gfCNCPoint1[13267] = {X 367.8420, Y 88.7408, Z -1.3333, A 0.000, B 0.000, C 0.000 }
gfCNCPoint1[13268] = {X 368.7992, Y 88.4188, Z -1.3333, A 0.000, B 0.000, C 0.000 }
gfCNCPoint1[13269] = {X 369.7143, Y 87.9916, Z -1.3333, A 0.000, B 0.000, C 0.000 }
gfCNCPoint1[13270] = {X 370.5758, Y 87.4644, Z -1.3333, A 0.000, B 0.000, C 0.000 }
gfCNCPoint1[13271] = {X 370.7919, Y 87.2394, Z -1.3333, A 0.000, B 0.000, C 0.000 }
gfCNCPoint1[13272] = {X 370.9033, Y 86.9481, Z -1.3333, A 0.000, B 0.000, C 0.000 }
gfCNCPoint1[13273] = {X 371.0969, Y 85.3932, Z -1.3333, A 0.000, B 0.000, C 0.000 }
gfCNCPoint1[13274] = {X 371.1614, Y 83.8276, Z -1.3333, A 0.000, B 0.000, C 0.000 }
gfCNCPoint1[13275] = {X 371.1611, Y 62.9983, Z -1.3333, A 0.000, B 0.000, C 0.000 }
gfCNCPoint1[13276] = {X 371.0248, Y 62.9840, Z -1.3333, A 0.000, B 0.000, C 0.000 }
gfCNCPoint1[13277] = {X 370.8891, Y 62.9651, Z -1.3333, A 0.000, B 0.000, C 0.000 }
gfCNCPoint1[13278] = {X 369.9694, Y 62.7082, Z -1.3333, A 0.000, B 0.000, C 0.000 }
gfCNCPoint1[13279] = {X 369.1346, Y 62.2446, Z -1.3333, A 0.000, B 0.000, C 0.000 }
gfCNCPoint1[13280] = {X 368.4305, Y 61.5997, Z -1.3333, A 0.000, B 0.000, C 0.000 }
gfCNCPoint1[13281] = {X 367.8955, Y 60.8087, Z -1.3333, A 0.000, B 0.000, C 0.000 }
gfCNCPoint1[13282] = {X 367.5590, Y 59.9151, Z -1.3333, A 0.000, B 0.000, C 0.000 }
gfCNCPoint1[13283] = {X 367.4394, Y 58.9678, Z -1.3333, A 0.000, B 0.000, C 0.000 }
gfCNCPoint1[13284] = {X 367.4393, Y 58.0000, Z -1.3333, A 0.000, B 0.000, C 0.000 }
gfCNCPoint1[13285] = {X 367.5416, Y 57.0921, Z -1.3333, A 0.000, B 0.000, C 0.000 }
gfCNCPoint1[13286] = {X 367.8433, Y 56.2298, Z -1.3333, A 0.000, B 0.000, C 0.000 }
gfCNCPoint1[13287] = {X 368.3294, Y 55.4562, Z -1.3333, A 0.000, B 0.000, C 0.000 }
gfCNCPoint1[13288] = {X 368.9754, Y 54.8101, Z -1.3333, A 0.000, B 0.000, C 0.000 }
gfCNCPoint1[13289] = {X 369.7490, Y 54.3240, Z -1.3333, A 0.000, B 0.000, C 0.000 }
gfCNCPoint1[13290] = {X 370.6114, Y 54.0223, Z -1.3333, A 0.000, B 0.000, C 0.000 }
gfCNCPoint1[13291] = {X 371.5193, Y 53.9200, Z -1.3333, A 0.000, B 0.000, C 0.000 }
gfCNCPoint1[13292] = {X 388.0597, Y 53.9200, Z -1.3333, A 0.000, B 0.000, C 0.000 }
gfCNCPoint1[13293] = {X 388.9676, Y 54.0223, Z -1.3333, A 0.000, B 0.000, C 0.000 }
gfCNCPoint1[13294] = {X 389.8299, Y 54.3240, Z -1.3333, A 0.000, B 0.000, C 0.000 }
gfCNCPoint1[13295] = {X 390.6035, Y 54.8101, Z -1.3333, A 0.000, B 0.000, C 0.000 }
gfCNCPoint1[13296] = {X 391.2496, Y 55.4562, Z -1.3333, A 0.000, B 0.000, C 0.000 }
gfCNCPoint1[13297] = {X 391.7356, Y 56.2298, Z -1.3333, A 0.000, B 0.000, C 0.000 }
gfCNCPoint1[13298] = {X 392.0374, Y 57.0921, Z -1.3333, A 0.000, B 0.000, C 0.000 }
gfCNCPoint1[13299] = {X 392.1397, Y 58.0000, Z -1.3333, A 0.000, B 0.000, C 0.000 }
gfCNCPoint1[13300] = {X 392.1397, Y 58.9342, Z -1.3333, A 0.000, B 0.000, C 0.000 }
gfCNCPoint1[13301] = {X 392.0298, Y 59.8744, Z -1.3333, A 0.000, B 0.000, C 0.000 }
gfCNCPoint1[13302] = {X 391.7063, Y 60.7639, Z -1.3333, A 0.000, B 0.000, C 0.000 }
gfCNCPoint1[13303] = {X 391.1724, Y 61.5726, Z -1.3333, A 0.000, B 0.000, C 0.000 }
gfCNCPoint1[13304] = {X 390.4636, Y 62.2335, Z -1.3333, A 0.000, B 0.000, C 0.000 }
gfCNCPoint1[13305] = {X 389.6195, Y 62.7095, Z -1.3333, A 0.000, B 0.000, C 0.000 }
gfCNCPoint1[13306] = {X 388.6872, Y 62.9742, Z -1.3333, A 0.000, B 0.000, C 0.000 }
gfCNCPoint1[13307] = {X 388.5540, Y 62.9932, Z -1.3333, A 0.000, B 0.000, C 0.000 }
gfCNCPoint1[13308] = {X 388.4202, Y 63.0078, Z -1.3333, A 0.000, B 0.000, C 0.000 }
gfCNCPoint1[13309] = {X 388.4176, Y 63.1548, Z -1.3333, A 0.000, B 0.000, C 0.000 }
gfCNCPoint1[13310] = {X 388.4156, Y 84.6157, Z -1.3333, A 0.000, B 0.000, C 0.000 }
gfCNCPoint1[13311] = {X 388.3564, Y 86.2534, Z -1.3333, A 0.000, B 0.000, C 0.000 }
gfCNCPoint1[13312] = {X 388.1546, Y 87.8797, Z -1.3333, A 0.000, B 0.000, C 0.000 }
gfCNCPoint1[13313] = {X 387.8118, Y 89.4822, Z -1.3333, A 0.000, B 0.000, C 0.000 }
gfCNCPoint1[13314] = {X 387.2905, Y 91.0377, Z -1.3333, A 0.000, B 0.000, C 0.000 }
gfCNCPoint1[13315] = {X 386.5561, Y 92.5046, Z -1.3333, A 0.000, B 0.000, C 0.000 }
gfCNCPoint1[13316] = {X 385.6232, Y 93.8539, Z -1.3333, A 0.000, B 0.000, C 0.000 }
gfCNCPoint1[13317] = {X 384.5101, Y 95.0589, Z -1.3333, A 0.000, B 0.000, C 0.000 }
gfCNCPoint1[13318] = {X 383.0155, Y 96.3179, Z -1.3333, A 0.000, B 0.000, C 0.000 }
gfCNCPoint1[13319] = {X 381.3959, Y 97.4112, Z -1.3333, A 0.000, B 0.000, C 0.000 }
gfCNCPoint1[13320] = {X 379.6694, Y 98.3265, Z -1.3333, A 0.000, B 0.000, C 0.000 }
gfCNCPoint1[13321] = {X 377.4145, Y 99.2771, Z -1.3333, A 0.000, B 0.000, C 0.000 }
gfCNCPoint1[13322] = {X 375.0967, Y 100.0618, Z -1.3333, A 0.000, B 0.000, C 0.000 }
gfCNCPoint1[13323] = {X 372.7281, Y 100.6767, Z -1.3333, A 0.000, B 0.000, C 0.000 }
gfCNCPoint1[13324] = {X 368.9280, Y 101.4118, Z -1.3333, A 0.000, B 0.000, C 0.000 }
gfCNCPoint1[13325] = {X 365.0969, Y 101.9635, Z -1.3333, A 0.000, B 0.000, C 0.000 }
gfCNCPoint1[13326] = {X 361.2438, Y 102.3303, Z -1.3333, A 0.000, B 0.000, C 0.000 }
gfCNCPoint1[13327] = {X 357.2421, Y 102.5707, Z -1.3333, A 0.000, B 0.000, C 0.000 }
gfCNCPoint1[13328] = {X 353.2361, Y 102.7240, Z -1.3333, A 0.000, B 0.000, C 0.000 }
gfCNCPoint1[13329] = {X 353.3455, Y 106.7225, Z -1.3333, A 0.000, B 0.000, C 0.000 }
gfCNCPoint1[13330] = {X 353.2339, Y 102.6440, Z -1.3333, A 0.000, B 0.000, C 0.000 }
gfCNCPoint1[13331] = {X 347.7211, Y 102.7124, Z -1.3333, A 0.000, B 0.000, C 0.000 }
gfCNCPoint1[13332] = {X 342.2087, Y 102.6158, Z -1.3333, A 0.000, B 0.000, C 0.000 }
gfCNCPoint1[13333] = {X 336.7017, Y 102.3544, Z -1.3333, A 0.000, B 0.000, C 0.000 }
gfCNCPoint1[13334] = {X 333.2238, Y 102.0803, Z -1.3333, A 0.000, B 0.000, C 0.000 }
gfCNCPoint1[13335] = {X 329.7596, Y 101.6688, Z -1.3333, A 0.000, B 0.000, C 0.000 }
gfCNCPoint1[13336] = {X 326.3144, Y 101.1205, Z -1.3333, A 0.000, B 0.000, C 0.000 }
gfCNCPoint1[13337] = {X 323.4875, Y 100.5209, Z -1.3333, A 0.000, B 0.000, C 0.000 }
gfCNCPoint1[13338] = {X 320.7125, Y 99.7145, Z -1.3333, A 0.000, B 0.000, C 0.000 }
gfCNCPoint1[13339] = {X 318.0046, Y 98.7056, Z -1.3333, A 0.000, B 0.000, C 0.000 }
gfCNCPoint1[13340] = {X 316.5155, Y 98.0196, Z -1.3333, A 0.000, B 0.000, C 0.000 }
gfCNCPoint1[13341] = {X 315.0892, Y 97.2110, Z -1.3333, A 0.000, B 0.000, C 0.000 }
gfCNCPoint1[13342] = {X 313.7357, Y 96.2857, Z -1.3333, A 0.000, B 0.000, C 0.000 }
gfCNCPoint1[13343] = {X 312.4647, Y 95.2501, Z -1.3333, A 0.000, B 0.000, C 0.000 }
gfCNCPoint1[13344] = {X 311.4884, Y 94.2784, Z -1.3333, A 0.000, B 0.000, C 0.000 }
gfCNCPoint1[13345] = {X 310.6340, Y 93.1980, Z -1.3333, A 0.000, B 0.000, C 0.000 }
gfCNCPoint1[13346] = {X 309.9137, Y 92.0239, Z -1.3333, A 0.000, B 0.000, C 0.000 }
gfCNCPoint1[13347] = {X 309.3376, Y 90.7727, Z -1.3333, A 0.000, B 0.000, C 0.000 }
gfCNCPoint1[13348] = {X 308.9138, Y 89.4621, Z -1.3333, A 0.000, B 0.000, C 0.000 }
gfCNCPoint1[13349] = {X 308.5760, Y 87.8658, Z -1.3333, A 0.000, B 0.000, C 0.000 }
gfCNCPoint1[13350] = {X 308.3765, Y 86.2464, Z -1.3333, A 0.000, B 0.000, C 0.000 }
gfCNCPoint1[13351] = {X 308.3167, Y 84.6159, Z -1.3333, A 0.000, B 0.000, C 0.000 }
gfCNCPoint1[13352] = {X 308.3180, Y 83.2313, Z -1.3333, A 0.000, B 0.000, C 0.000 }
gfCNCPoint1[13353] = {X 308.3180, Y 62.9244, Z -1.3333, A 0.000, B 0.000, C 0.000 }
gfCNCPoint1[13354] = {X 307.4752, Y 62.7738, Z -1.3333, A 0.000, B 0.000, C 0.000 }
gfCNCPoint1[13355] = {X 306.6837, Y 62.4472, Z -1.3333, A 0.000, B 0.000, C 0.000 }
gfCNCPoint1[13356] = {X 305.9799, Y 61.9597, Z -1.3333, A 0.000, B 0.000, C 0.000 }
gfCNCPoint1[13357] = {X 305.3959, Y 61.3336, Z -1.3333, A 0.000, B 0.000, C 0.000 }
gfCNCPoint1[13358] = {X 304.9585, Y 60.5976, Z -1.3333, A 0.000, B 0.000, C 0.000 }
gfCNCPoint1[13359] = {X 304.6878, Y 59.7853, Z -1.3333, A 0.000, B 0.000, C 0.000 }
gfCNCPoint1[13360] = {X 304.5962, Y 58.9340, Z -1.3333, A 0.000, B 0.000, C 0.000 }
gfCNCPoint1[13361] = {X 304.5962, Y 58.0000, Z -1.3333, A 0.000, B 0.000, C 0.000 }
gfCNCPoint1[13362] = {X 304.6965, Y 57.1099, Z -1.3333, A 0.000, B 0.000, C 0.000 }
gfCNCPoint1[13363] = {X 304.9923, Y 56.2645, Z -1.3333, A 0.000, B 0.000, C 0.000 }
gfCNCPoint1[13364] = {X 305.4689, Y 55.5060, Z -1.3333, A 0.000, B 0.000, C 0.000 }
gfCNCPoint1[13365] = {X 306.1023, Y 54.8727, Z -1.3333, A 0.000, B 0.000, C 0.000 }
gfCNCPoint1[13366] = {X 306.8607, Y 54.3961, Z -1.3333, A 0.000, B 0.000, C 0.000 }
gfCNCPoint1[13367] = {X 307.7061, Y 54.1003, Z -1.3333, A 0.000, B 0.000, C 0.000 }
gfCNCPoint1[13368] = {X 308.5962, Y 54.0000, Z -1.3333, A 0.000, B 0.000, C 0.000 }
gfCNCPoint1[13369] = {X 324.3107, Y 54.0000, Z -1.3333, A 0.000, B 0.000, C 0.000 }
gfCNCPoint1[13370] = {X 325.2008, Y 54.1003, Z -1.3333, A 0.000, B 0.000, C 0.000 }
gfCNCPoint1[13371] = {X 326.0462, Y 54.3961, Z -1.3333, A 0.000, B 0.000, C 0.000 }
gfCNCPoint1[13372] = {X 326.8046, Y 54.8727, Z -1.3333, A 0.000, B 0.000, C 0.000 }
gfCNCPoint1[13373] = {X 327.4380, Y 55.5060, Z -1.3333, A 0.000, B 0.000, C 0.000 }
gfCNCPoint1[13374] = {X 327.9146, Y 56.2645, Z -1.3333, A 0.000, B 0.000, C 0.000 }
gfCNCPoint1[13375] = {X 328.2104, Y 57.1099, Z -1.3333, A 0.000, B 0.000, C 0.000 }
gfCNCPoint1[13376] = {X 328.3107, Y 58.0000, Z -1.3333, A 0.000, B 0.000, C 0.000 }
gfCNCPoint1[13377] = {X 328.3107, Y 58.9341, Z -1.3333, A 0.000, B 0.000, C 0.000 }
gfCNCPoint1[13378] = {X 328.2147, Y 59.7843, Z -1.3333, A 0.000, B 0.000, C 0.000 }
gfCNCPoint1[13379] = {X 327.9419, Y 60.5952, Z -1.3333, A 0.000, B 0.000, C 0.000 }
gfCNCPoint1[13380] = {X 327.5044, Y 61.3305, Z -1.3333, A 0.000, B 0.000, C 0.000 }
gfCNCPoint1[13381] = {X 326.9218, Y 61.9572, Z -1.3333, A 0.000, B 0.000, C 0.000 }
gfCNCPoint1[13382] = {X 326.2204, Y 62.4471, Z -1.3333, A 0.000, B 0.000, C 0.000 }
gfCNCPoint1[13383] = {X 325.4315, Y 62.7783, Z -1.3333, A 0.000, B 0.000, C 0.000 }
gfCNCPoint1[13384] = {X 324.5905, Y 62.9360, Z -1.3333, A 0.000, B 0.000, C 0.000 }
gfCNCPoint1[13385] = {X 324.5919, Y 83.2313, Z -1.3333, A 0.000, B 0.000, C 0.000 }
gfCNCPoint1[13386] = {X 324.6054, Y 84.6159, Z -1.3333, A 0.000, B 0.000, C 0.000 }
gfCNCPoint1[13387] = {X 324.6887, Y 85.9184, Z -1.3333, A 0.000, B 0.000, C 0.000 }
gfCNCPoint1[13388] = {X 324.9294, Y 87.2011, Z -1.3333, A 0.000, B 0.000, C 0.000 }
gfCNCPoint1[13389] = {X 325.2359, Y 87.5559, Z -1.3333, A 0.000, B 0.000, C 0.000 }
gfCNCPoint1[13390] = {X 325.6219, Y 87.8220, Z -1.3333, A 0.000, B 0.000, C 0.000 }
gfCNCPoint1[13391] = {X 326.0749, Y 88.0775, Z -1.3333, A 0.000, B 0.000, C 0.000 }
gfCNCPoint1[13392] = {X 327.5502, Y 88.6916, Z -1.3333, A 0.000, B 0.000, C 0.000 }
gfCNCPoint1[13393] = {X 329.0843, Y 89.1390, Z -1.3333, A 0.000, B 0.000, C 0.000 }
gfCNCPoint1[13394] = {X 332.1822, Y 89.7592, Z -1.3333, A 0.000, B 0.000, C 0.000 }
gfCNCPoint1[13395] = {X 335.3167, Y 90.1542, Z -1.3333, A 0.000, B 0.000, C 0.000 }
gfCNCPoint1[13396] = {X 340.5042, Y 90.5381, Z -1.3333, A 0.000, B 0.000, C 0.000 }
gfCNCPoint1[13397] = {X 345.7039, Y 90.6832, Z -1.3333, A 0.000, B 0.000, C 0.000 }
gfCNCPoint1[13398] = {X 350.5564, Y 90.6891, Z -1.3333, A 0.000, B 0.000, C 0.000 }
gfCNCPoint1[13399] = {X 355.4059, Y 90.5203, Z -1.3333, A 0.000, B 0.000, C 0.000 }
gfCNCPoint1[13400] = {X 360.2461, Y 90.1768, Z -1.3333, A 0.000, B 0.000, C 0.000 }
gfCNCPoint1[13401] = {X 362.8123, Y 89.8853, Z -1.3333, A 0.000, B 0.000, C 0.000 }
gfCNCPoint1[13402] = {X 365.3548, Y 89.4317, Z -1.3333, A 0.000, B 0.000, C 0.000 }
gfCNCPoint1[13403] = {X 367.8634, Y 88.8179, Z -1.3333, A 0.000, B 0.000, C 0.000 }
gfCNCPoint1[13404] = {X 368.8291, Y 88.4930, Z -1.3333, A 0.000, B 0.000, C 0.000 }
gfCNCPoint1[13405] = {X 369.7523, Y 88.0620, Z -1.3333, A 0.000, B 0.000, C 0.000 }
gfCNCPoint1[13406] = {X 370.6213, Y 87.5302, Z -1.3333, A 0.000, B 0.000, C 0.000 }
gfCNCPoint1[13407] = {X 370.8594, Y 87.2823, Z -1.3333, A 0.000, B 0.000, C 0.000 }
gfCNCPoint1[13408] = {X 370.9822, Y 86.9612, Z -1.3333, A 0.000, B 0.000, C 0.000 }
gfCNCPoint1[13409] = {X 371.1766, Y 85.3997, Z -1.3333, A 0.000, B 0.000, C 0.000 }
gfCNCPoint1[13410] = {X 371.2414, Y 83.8276, Z -1.3333, A 0.000, B 0.000, C 0.000 }
gfCNCPoint1[13411] = {X 371.2396, Y 63.0383, Z -1.3333, A 0.000, B 0.000, C 0.000 }
gfCNCPoint1[13412] = {X 371.2440, Y 62.9246, Z -1.3333, A 0.000, B 0.000, C 0.000 }
gfCNCPoint1[13413] = {X 371.0723, Y 62.9090, Z -1.3333, A 0.000, B 0.000, C 0.000 }
gfCNCPoint1[13414] = {X 370.9014, Y 62.8861, Z -1.3333, A 0.000, B 0.000, C 0.000 }
gfCNCPoint1[13415] = {X 369.9947, Y 62.6321, Z -1.3333, A 0.000, B 0.000, C 0.000 }
gfCNCPoint1[13416] = {X 369.1724, Y 62.1733, Z -1.3333, A 0.000, B 0.000, C 0.000 }
gfCNCPoint1[13417] = {X 368.4802, Y 61.5349, Z -1.3333, A 0.000, B 0.000, C 0.000 }
gfCNCPoint1[13418] = {X 367.9565, Y 60.7524, Z -1.3333, A 0.000, B 0.000, C 0.000 }
gfCNCPoint1[13419] = {X 367.6301, Y 59.8691, Z -1.3333, A 0.000, B 0.000, C 0.000 }
gfCNCPoint1[13420] = {X 367.5193, Y 58.9340, Z -1.3333, A 0.000, B 0.000, C 0.000 }
gfCNCPoint1[13421] = {X 367.5193, Y 58.0000, Z -1.3333, A 0.000, B 0.000, C 0.000 }
gfCNCPoint1[13422] = {X 367.6196, Y 57.1099, Z -1.3333, A 0.000, B 0.000, C 0.000 }
gfCNCPoint1[13423] = {X 367.9154, Y 56.2645, Z -1.3333, A 0.000, B 0.000, C 0.000 }
gfCNCPoint1[13424] = {X 368.3920, Y 55.5060, Z -1.3333, A 0.000, B 0.000, C 0.000 }
gfCNCPoint1[13425] = {X 369.0253, Y 54.8727, Z -1.3333, A 0.000, B 0.000, C 0.000 }
gfCNCPoint1[13426] = {X 369.7837, Y 54.3961, Z -1.3333, A 0.000, B 0.000, C 0.000 }
gfCNCPoint1[13427] = {X 370.6292, Y 54.1003, Z -1.3333, A 0.000, B 0.000, C 0.000 }
gfCNCPoint1[13428] = {X 371.5193, Y 54.0000, Z -1.3333, A 0.000, B 0.000, C 0.000 }
gfCNCPoint1[13429] = {X 388.0597, Y 54.0000, Z -1.3333, A 0.000, B 0.000, C 0.000 }
gfCNCPoint1[13430] = {X 388.9498, Y 54.1003, Z -1.3333, A 0.000, B 0.000, C 0.000 }
gfCNCPoint1[13431] = {X 389.7952, Y 54.3961, Z -1.3333, A 0.000, B 0.000, C 0.000 }
gfCNCPoint1[13432] = {X 390.5536, Y 54.8727, Z -1.3333, A 0.000, B 0.000, C 0.000 }
gfCNCPoint1[13433] = {X 391.1870, Y 55.5060, Z -1.3333, A 0.000, B 0.000, C 0.000 }
gfCNCPoint1[13434] = {X 391.6636, Y 56.2645, Z -1.3333, A 0.000, B 0.000, C 0.000 }
gfCNCPoint1[13435] = {X 391.9594, Y 57.1099, Z -1.3333, A 0.000, B 0.000, C 0.000 }
gfCNCPoint1[13436] = {X 392.0597, Y 58.0000, Z -1.3333, A 0.000, B 0.000, C 0.000 }
gfCNCPoint1[13437] = {X 392.0595, Y 58.9671, Z -1.3333, A 0.000, B 0.000, C 0.000 }
gfCNCPoint1[13438] = {X 391.9482, Y 59.8719, Z -1.3333, A 0.000, B 0.000, C 0.000 }
gfCNCPoint1[13439] = {X 391.6348, Y 60.7280, Z -1.3333, A 0.000, B 0.000, C 0.000 }
gfCNCPoint1[13440] = {X 391.1113, Y 61.5210, Z -1.3333, A 0.000, B 0.000, C 0.000 }
gfCNCPoint1[13441] = {X 390.4163, Y 62.1689, Z -1.3333, A 0.000, B 0.000, C 0.000 }
gfCNCPoint1[13442] = {X 389.5887, Y 62.6357, Z -1.3333, A 0.000, B 0.000, C 0.000 }
gfCNCPoint1[13443] = {X 388.6746, Y 62.8952, Z -1.3333, A 0.000, B 0.000, C 0.000 }
gfCNCPoint1[13444] = {X 388.5085, Y 62.9182, Z -1.3333, A 0.000, B 0.000, C 0.000 }
gfCNCPoint1[13445] = {X 388.3415, Y 62.9342, Z -1.3333, A 0.000, B 0.000, C 0.000 }
gfCNCPoint1[13446] = {X 388.3376, Y 63.1540, Z -1.3333, A 0.000, B 0.000, C 0.000 }
gfCNCPoint1[13447] = {X 388.3376, Y 83.9236, Z -1.3333, A 0.000, B 0.000, C 0.000 }
gfCNCPoint1[13448] = {X 388.3356, Y 84.6159, Z -1.3333, A 0.000, B 0.000, C 0.000 }
gfCNCPoint1[13449] = {X 388.2766, Y 86.2468, Z -1.3333, A 0.000, B 0.000, C 0.000 }
gfCNCPoint1[13450] = {X 388.0757, Y 87.8663, Z -1.3333, A 0.000, B 0.000, C 0.000 }
gfCNCPoint1[13451] = {X 387.7344, Y 89.4621, Z -1.3333, A 0.000, B 0.000, C 0.000 }
gfCNCPoint1[13452] = {X 387.2167, Y 91.0069, Z -1.3333, A 0.000, B 0.000, C 0.000 }
gfCNCPoint1[13453] = {X 386.4873, Y 92.4638, Z -1.3333, A 0.000, B 0.000, C 0.000 }
gfCNCPoint1[13454] = {X 385.5607, Y 93.8039, Z -1.3333, A 0.000, B 0.000, C 0.000 }
gfCNCPoint1[13455] = {X 384.4553, Y 95.0007, Z -1.3333, A 0.000, B 0.000, C 0.000 }
gfCNCPoint1[13456] = {X 382.9672, Y 96.2541, Z -1.3333, A 0.000, B 0.000, C 0.000 }
gfCNCPoint1[13457] = {X 381.3546, Y 97.3426, Z -1.3333, A 0.000, B 0.000, C 0.000 }
gfCNCPoint1[13458] = {X 379.6357, Y 98.2540, Z -1.3333, A 0.000, B 0.000, C 0.000 }
gfCNCPoint1[13459] = {X 377.3861, Y 99.2023, Z -1.3333, A 0.000, B 0.000, C 0.000 }
gfCNCPoint1[13460] = {X 375.0738, Y 99.9852, Z -1.3333, A 0.000, B 0.000, C 0.000 }
gfCNCPoint1[13461] = {X 372.7108, Y 100.5986, Z -1.3333, A 0.000, B 0.000, C 0.000 }
gfCNCPoint1[13462] = {X 368.9146, Y 101.3330, Z -1.3333, A 0.000, B 0.000, C 0.000 }
gfCNCPoint1[13463] = {X 365.0874, Y 101.8841, Z -1.3333, A 0.000, B 0.000, C 0.000 }
gfCNCPoint1[13464] = {X 361.2381, Y 102.2505, Z -1.3333, A 0.000, B 0.000, C 0.000 }
gfCNCPoint1[13465] = {X 357.2381, Y 102.4908, Z -1.3333, A 0.000, B 0.000, C 0.000 }
gfCNCPoint1[13466] = {X 353.2339, Y 102.6440, Z -1.3333, A 0.000, B 0.000, C 0.000 }
gfCNCPoint1[13467] = {X 353.3455, Y 106.7225, Z -1.3333, A 0.000, B 0.000, C 0.000 }
gfCNCPoint1[13468] = {X 353.3455, Y 106.7225, Z 1.6667, A 0.000, B 0.000, C 0.000 }
gfCNCPoint1[13469] = {X 353.3455, Y 106.7225, Z 11.0000, A 0.000, B 0.000, C 0.000 }
gfCNCPoint1[13470] = {X 411.5994, Y 79.5934, Z 11.0000, A 0.000, B 0.000, C 0.000 }
gfCNCPoint1[13471] = {X 411.5994, Y 79.5934, Z 1.6667, A 0.000, B 0.000, C 0.000 }
gfCNCPoint1[13472] = {X 411.5994, Y 79.5934, Z -1.3333, A 0.000, B 0.000, C 0.000 }
gfCNCPoint1[13473] = {X 413.7997, Y 83.0292, Z -1.3333, A 0.000, B 0.000, C 0.000 }
gfCNCPoint1[13474] = {X 428.0558, Y 73.8994, Z -1.3333, A 0.000, B 0.000, C 0.000 }
gfCNCPoint1[13475] = {X 403.7554, Y 64.3645, Z -1.3333, A 0.000, B 0.000, C 0.000 }
gfCNCPoint1[13476] = {X 402.0597, Y 63.8030, Z -1.3333, A 0.000, B 0.000, C 0.000 }
gfCNCPoint1[13477] = {X 400.3124, Y 63.4313, Z -1.3333, A 0.000, B 0.000, C 0.000 }
gfCNCPoint1[13478] = {X 398.5349, Y 63.2540, Z -1.3333, A 0.000, B 0.000, C 0.000 }
gfCNCPoint1[13479] = {X 397.5823, Y 63.1425, Z -1.3333, A 0.000, B 0.000, C 0.000 }
gfCNCPoint1[13480] = {X 396.6778, Y 62.8236, Z -1.3333, A 0.000, B 0.000, C 0.000 }
gfCNCPoint1[13481] = {X 395.8660, Y 62.3130, Z -1.3333, A 0.000, B 0.000, C 0.000 }
gfCNCPoint1[13482] = {X 395.1868, Y 61.6358, Z -1.3333, A 0.000, B 0.000, C 0.000 }
gfCNCPoint1[13483] = {X 394.6738, Y 60.8255, Z -1.3333, A 0.000, B 0.000, C 0.000 }
gfCNCPoint1[13484] = {X 394.3522, Y 59.9220, Z -1.3333, A 0.000, B 0.000, C 0.000 }
gfCNCPoint1[13485] = {X 394.2379, Y 58.9697, Z -1.3333, A 0.000, B 0.000, C 0.000 }
gfCNCPoint1[13486] = {X 394.2377, Y 58.0000, Z -1.3333, A 0.000, B 0.000, C 0.000 }
gfCNCPoint1[13487] = {X 394.3460, Y 57.0387, Z -1.3333, A 0.000, B 0.000, C 0.000 }
gfCNCPoint1[13488] = {X 394.6655, Y 56.1256, Z -1.3333, A 0.000, B 0.000, C 0.000 }
gfCNCPoint1[13489] = {X 395.1802, Y 55.3065, Z -1.3333, A 0.000, B 0.000, C 0.000 }
gfCNCPoint1[13490] = {X 395.8642, Y 54.6225, Z -1.3333, A 0.000, B 0.000, C 0.000 }
gfCNCPoint1[13491] = {X 396.6833, Y 54.1078, Z -1.3333, A 0.000, B 0.000, C 0.000 }
gfCNCPoint1[13492] = {X 397.5964, Y 53.7883, Z -1.3333, A 0.000, B 0.000, C 0.000 }
gfCNCPoint1[13493] = {X 398.5577, Y 53.6800, Z -1.3333, A 0.000, B 0.000, C 0.000 }
gfCNCPoint1[13494] = {X 419.4886, Y 53.6800, Z -1.3333, A 0.000, B 0.000, C 0.000 }
gfCNCPoint1[13495] = {X 420.4499, Y 53.7883, Z -1.3333, A 0.000, B 0.000, C 0.000 }
gfCNCPoint1[13496] = {X 421.3630, Y 54.1078, Z -1.3333, A 0.000, B 0.000, C 0.000 }
gfCNCPoint1[13497] = {X 422.1821, Y 54.6225, Z -1.3333, A 0.000, B 0.000, C 0.000 }
gfCNCPoint1[13498] = {X 422.8661, Y 55.3065, Z -1.3333, A 0.000, B 0.000, C 0.000 }
gfCNCPoint1[13499] = {X 423.3808, Y 56.1256, Z -1.3333, A 0.000, B 0.000, C 0.000 }
gfCNCPoint1[13500] = {X 423.7003, Y 57.0387, Z -1.3333, A 0.000, B 0.000, C 0.000 }
gfCNCPoint1[13501] = {X 423.8086, Y 58.0000, Z -1.3333, A 0.000, B 0.000, C 0.000 }
gfCNCPoint1[13502] = {X 423.8086, Y 58.2329, Z -1.3333, A 0.000, B 0.000, C 0.000 }
gfCNCPoint1[13503] = {X 429.6116, Y 60.4947, Z -1.3333, A 0.000, B 0.000, C 0.000 }
gfCNCPoint1[13504] = {X 457.8614, Y 71.7026, Z -1.3333, A 0.000, B 0.000, C 0.000 }
gfCNCPoint1[13505] = {X 457.8614, Y 63.2124, Z -1.3333, A 0.000, B 0.000, C 0.000 }
gfCNCPoint1[13506] = {X 457.0096, Y 63.0035, Z -1.3333, A 0.000, B 0.000, C 0.000 }
gfCNCPoint1[13507] = {X 456.2176, Y 62.6267, Z -1.3333, A 0.000, B 0.000, C 0.000 }
gfCNCPoint1[13508] = {X 455.5180, Y 62.0978, Z -1.3333, A 0.000, B 0.000, C 0.000 }
gfCNCPoint1[13509] = {X 454.9396, Y 61.4384, Z -1.3333, A 0.000, B 0.000, C 0.000 }
gfCNCPoint1[13510] = {X 454.5063, Y 60.6759, Z -1.3333, A 0.000, B 0.000, C 0.000 }
gfCNCPoint1[13511] = {X 454.2360, Y 59.8415, Z -1.3333, A 0.000, B 0.000, C 0.000 }
gfCNCPoint1[13512] = {X 454.1398, Y 58.9697, Z -1.3333, A 0.000, B 0.000, C 0.000 }
gfCNCPoint1[13513] = {X 454.1396, Y 58.0000, Z -1.3333, A 0.000, B 0.000, C 0.000 }
gfCNCPoint1[13514] = {X 454.2479, Y 57.0387, Z -1.3333, A 0.000, B 0.000, C 0.000 }
gfCNCPoint1[13515] = {X 454.5674, Y 56.1256, Z -1.3333, A 0.000, B 0.000, C 0.000 }
gfCNCPoint1[13516] = {X 455.0821, Y 55.3065, Z -1.3333, A 0.000, B 0.000, C 0.000 }
gfCNCPoint1[13517] = {X 455.7661, Y 54.6225, Z -1.3333, A 0.000, B 0.000, C 0.000 }
gfCNCPoint1[13518] = {X 456.5852, Y 54.1078, Z -1.3333, A 0.000, B 0.000, C 0.000 }
gfCNCPoint1[13519] = {X 457.4983, Y 53.7883, Z -1.3333, A 0.000, B 0.000, C 0.000 }
gfCNCPoint1[13520] = {X 458.4596, Y 53.6800, Z -1.3333, A 0.000, B 0.000, C 0.000 }
gfCNCPoint1[13521] = {X 475.0000, Y 53.6800, Z -1.3333, A 0.000, B 0.000, C 0.000 }
gfCNCPoint1[13522] = {X 475.9613, Y 53.7883, Z -1.3333, A 0.000, B 0.000, C 0.000 }
gfCNCPoint1[13523] = {X 476.8744, Y 54.1078, Z -1.3333, A 0.000, B 0.000, C 0.000 }
gfCNCPoint1[13524] = {X 477.6935, Y 54.6225, Z -1.3333, A 0.000, B 0.000, C 0.000 }
gfCNCPoint1[13525] = {X 478.3775, Y 55.3065, Z -1.3333, A 0.000, B 0.000, C 0.000 }
gfCNCPoint1[13526] = {X 478.8922, Y 56.1256, Z -1.3333, A 0.000, B 0.000, C 0.000 }
gfCNCPoint1[13527] = {X 479.2117, Y 57.0387, Z -1.3333, A 0.000, B 0.000, C 0.000 }
gfCNCPoint1[13528] = {X 479.3200, Y 58.0000, Z -1.3333, A 0.000, B 0.000, C 0.000 }
gfCNCPoint1[13529] = {X 479.3200, Y 58.9342, Z -1.3333, A 0.000, B 0.000, C 0.000 }
gfCNCPoint1[13530] = {X 479.2299, Y 59.8116, Z -1.3333, A 0.000, B 0.000, C 0.000 }
gfCNCPoint1[13531] = {X 478.9636, Y 60.6524, Z -1.3333, A 0.000, B 0.000, C 0.000 }
gfCNCPoint1[13532] = {X 478.5320, Y 61.4215, Z -1.3333, A 0.000, B 0.000, C 0.000 }
gfCNCPoint1[13533] = {X 477.9532, Y 62.0870, Z -1.3333, A 0.000, B 0.000, C 0.000 }
gfCNCPoint1[13534] = {X 477.2513, Y 62.6211, Z -1.3333, A 0.000, B 0.000, C 0.000 }
gfCNCPoint1[13535] = {X 476.4556, Y 63.0014, Z -1.3333, A 0.000, B 0.000, C 0.000 }
gfCNCPoint1[13536] = {X 475.5992, Y 63.2123, Z -1.3333, A 0.000, B 0.000, C 0.000 }
gfCNCPoint1[13537] = {X 475.5996, Y 92.7691, Z -1.3333, A 0.000, B 0.000, C 0.000 }
gfCNCPoint1[13538] = {X 475.9955, Y 92.8681, Z -1.3333, A 0.000, B 0.000, C 0.000 }
gfCNCPoint1[13539] = {X 476.3859, Y 92.9874, Z -1.3333, A 0.000, B 0.000, C 0.000 }
gfCNCPoint1[13540] = {X 477.1980, Y 93.3562, Z -1.3333, A 0.000, B 0.000, C 0.000 }
gfCNCPoint1[13541] = {X 477.9164, Y 93.8849, Z -1.3333, A 0.000, B 0.000, C 0.000 }
gfCNCPoint1[13542] = {X 478.5101, Y 94.5506, Z -1.3333, A 0.000, B 0.000, C 0.000 }
gfCNCPoint1[13543] = {X 478.9535, Y 95.3245, Z -1.3333, A 0.000, B 0.000, C 0.000 }
gfCNCPoint1[13544] = {X 479.2274, Y 96.1734, Z -1.3333, A 0.000, B 0.000, C 0.000 }
gfCNCPoint1[13545] = {X 479.3200, Y 97.0605, Z -1.3333, A 0.000, B 0.000, C 0.000 }
gfCNCPoint1[13546] = {X 479.3200, Y 98.0000, Z -1.3333, A 0.000, B 0.000, C 0.000 }
gfCNCPoint1[13547] = {X 479.2117, Y 98.9613, Z -1.3333, A 0.000, B 0.000, C 0.000 }
gfCNCPoint1[13548] = {X 478.8922, Y 99.8744, Z -1.3333, A 0.000, B 0.000, C 0.000 }
gfCNCPoint1[13549] = {X 478.3775, Y 100.6935, Z -1.3333, A 0.000, B 0.000, C 0.000 }
gfCNCPoint1[13550] = {X 477.6935, Y 101.3775, Z -1.3333, A 0.000, B 0.000, C 0.000 }
gfCNCPoint1[13551] = {X 476.8744, Y 101.8922, Z -1.3333, A 0.000, B 0.000, C 0.000 }
gfCNCPoint1[13552] = {X 475.9613, Y 102.2117, Z -1.3333, A 0.000, B 0.000, C 0.000 }
gfCNCPoint1[13553] = {X 475.0000, Y 102.3200, Z -1.3333, A 0.000, B 0.000, C 0.000 }
gfCNCPoint1[13554] = {X 458.4596, Y 102.3200, Z -1.3333, A 0.000, B 0.000, C 0.000 }
gfCNCPoint1[13555] = {X 457.4983, Y 102.2117, Z -1.3333, A 0.000, B 0.000, C 0.000 }
gfCNCPoint1[13556] = {X 456.5852, Y 101.8922, Z -1.3333, A 0.000, B 0.000, C 0.000 }
gfCNCPoint1[13557] = {X 455.7661, Y 101.3775, Z -1.3333, A 0.000, B 0.000, C 0.000 }
gfCNCPoint1[13558] = {X 455.0821, Y 100.6935, Z -1.3333, A 0.000, B 0.000, C 0.000 }
gfCNCPoint1[13559] = {X 454.5674, Y 99.8744, Z -1.3333, A 0.000, B 0.000, C 0.000 }
gfCNCPoint1[13560] = {X 454.2479, Y 98.9613, Z -1.3333, A 0.000, B 0.000, C 0.000 }
gfCNCPoint1[13561] = {X 454.1396, Y 98.0000, Z -1.3333, A 0.000, B 0.000, C 0.000 }
gfCNCPoint1[13562] = {X 454.1396, Y 97.0659, Z -1.3333, A 0.000, B 0.000, C 0.000 }
gfCNCPoint1[13563] = {X 454.2295, Y 96.1891, Z -1.3333, A 0.000, B 0.000, C 0.000 }
gfCNCPoint1[13564] = {X 454.4955, Y 95.3488, Z -1.3333, A 0.000, B 0.000, C 0.000 }
gfCNCPoint1[13565] = {X 454.9265, Y 94.5800, Z -1.3333, A 0.000, B 0.000, C 0.000 }
gfCNCPoint1[13566] = {X 455.5046, Y 93.9147, Z -1.3333, A 0.000, B 0.000, C 0.000 }
gfCNCPoint1[13567] = {X 456.2057, Y 93.3805, Z -1.3333, A 0.000, B 0.000, C 0.000 }
gfCNCPoint1[13568] = {X 457.0006, Y 92.9998, Z -1.3333, A 0.000, B 0.000, C 0.000 }
gfCNCPoint1[13569] = {X 457.8563, Y 92.7883, Z -1.3333, A 0.000, B 0.000, C 0.000 }
gfCNCPoint1[13570] = {X 457.8563, Y 85.5950, Z -1.3333, A 0.000, B 0.000, C 0.000 }
gfCNCPoint1[13571] = {X 444.8578, Y 80.4996, Z -1.3333, A 0.000, B 0.000, C 0.000 }
gfCNCPoint1[13572] = {X 420.0225, Y 96.5880, Z -1.3333, A 0.000, B 0.000, C 0.000 }
gfCNCPoint1[13573] = {X 420.0267, Y 97.0645, Z -1.3333, A 0.000, B 0.000, C 0.000 }
gfCNCPoint1[13574] = {X 420.0267, Y 98.0000, Z -1.3333, A 0.000, B 0.000, C 0.000 }
gfCNCPoint1[13575] = {X 419.9184, Y 98.9613, Z -1.3333, A 0.000, B 0.000, C 0.000 }
gfCNCPoint1[13576] = {X 419.5989, Y 99.8744, Z -1.3333, A 0.000, B 0.000, C 0.000 }
gfCNCPoint1[13577] = {X 419.0842, Y 100.6935, Z -1.3333, A 0.000, B 0.000, C 0.000 }
gfCNCPoint1[13578] = {X 418.4002, Y 101.3775, Z -1.3333, A 0.000, B 0.000, C 0.000 }
gfCNCPoint1[13579] = {X 417.5811, Y 101.8922, Z -1.3333, A 0.000, B 0.000, C 0.000 }
gfCNCPoint1[13580] = {X 416.6680, Y 102.2117, Z -1.3333, A 0.000, B 0.000, C 0.000 }
gfCNCPoint1[13581] = {X 415.7067, Y 102.3200, Z -1.3333, A 0.000, B 0.000, C 0.000 }
gfCNCPoint1[13582] = {X 396.4059, Y 102.3200, Z -1.3333, A 0.000, B 0.000, C 0.000 }
gfCNCPoint1[13583] = {X 395.4447, Y 102.2117, Z -1.3333, A 0.000, B 0.000, C 0.000 }
gfCNCPoint1[13584] = {X 394.5316, Y 101.8922, Z -1.3333, A 0.000, B 0.000, C 0.000 }
gfCNCPoint1[13585] = {X 393.7125, Y 101.3775, Z -1.3333, A 0.000, B 0.000, C 0.000 }
gfCNCPoint1[13586] = {X 393.0284, Y 100.6935, Z -1.3333, A 0.000, B 0.000, C 0.000 }
gfCNCPoint1[13587] = {X 392.5138, Y 99.8744, Z -1.3333, A 0.000, B 0.000, C 0.000 }
gfCNCPoint1[13588] = {X 392.1943, Y 98.9613, Z -1.3333, A 0.000, B 0.000, C 0.000 }
gfCNCPoint1[13589] = {X 392.0859, Y 98.0000, Z -1.3333, A 0.000, B 0.000, C 0.000 }
gfCNCPoint1[13590] = {X 392.0859, Y 97.0659, Z -1.3333, A 0.000, B 0.000, C 0.000 }
gfCNCPoint1[13591] = {X 392.1938, Y 96.1068, Z -1.3333, A 0.000, B 0.000, C 0.000 }
gfCNCPoint1[13592] = {X 392.5118, Y 95.1956, Z -1.3333, A 0.000, B 0.000, C 0.000 }
gfCNCPoint1[13593] = {X 393.0242, Y 94.3777, Z -1.3333, A 0.000, B 0.000, C 0.000 }
gfCNCPoint1[13594] = {X 393.7054, Y 93.6940, Z -1.3333, A 0.000, B 0.000, C 0.000 }
gfCNCPoint1[13595] = {X 394.5214, Y 93.1786, Z -1.3333, A 0.000, B 0.000, C 0.000 }
gfCNCPoint1[13596] = {X 395.4315, Y 92.8573, Z -1.3333, A 0.000, B 0.000, C 0.000 }
gfCNCPoint1[13597] = {X 396.3902, Y 92.7460, Z -1.3333, A 0.000, B 0.000, C 0.000 }
gfCNCPoint1[13598] = {X 397.3435, Y 92.7059, Z -1.3333, A 0.000, B 0.000, C 0.000 }
gfCNCPoint1[13599] = {X 398.2933, Y 92.6157, Z -1.3333, A 0.000, B 0.000, C 0.000 }
gfCNCPoint1[13600] = {X 398.9443, Y 92.4580, Z -1.3333, A 0.000, B 0.000, C 0.000 }
gfCNCPoint1[13601] = {X 399.5436, Y 92.1590, Z -1.3333, A 0.000, B 0.000, C 0.000 }
gfCNCPoint1[13602] = {X 413.7997, Y 83.0292, Z -1.3333, A 0.000, B 0.000, C 0.000 }
gfCNCPoint1[13603] = {X 411.6425, Y 79.6607, Z -1.3333, A 0.000, B 0.000, C 0.000 }
gfCNCPoint1[13604] = {X 413.8429, Y 83.0966, Z -1.3333, A 0.000, B 0.000, C 0.000 }
gfCNCPoint1[13605] = {X 428.2310, Y 73.8822, Z -1.3333, A 0.000, B 0.000, C 0.000 }
gfCNCPoint1[13606] = {X 403.7847, Y 64.2900, Z -1.3333, A 0.000, B 0.000, C 0.000 }
gfCNCPoint1[13607] = {X 402.0801, Y 63.7256, Z -1.3333, A 0.000, B 0.000, C 0.000 }
gfCNCPoint1[13608] = {X 400.3237, Y 63.3521, Z -1.3333, A 0.000, B 0.000, C 0.000 }
gfCNCPoint1[13609] = {X 398.5369, Y 63.1740, Z -1.3333, A 0.000, B 0.000, C 0.000 }
gfCNCPoint1[13610] = {X 397.6017, Y 63.0649, Z -1.3333, A 0.000, B 0.000, C 0.000 }
gfCNCPoint1[13611] = {X 396.7137, Y 62.7521, Z -1.3333, A 0.000, B 0.000, C 0.000 }
gfCNCPoint1[13612] = {X 395.9166, Y 62.2510, Z -1.3333, A 0.000, B 0.000, C 0.000 }
gfCNCPoint1[13613] = {X 395.2497, Y 61.5863, Z -1.3333, A 0.000, B 0.000, C 0.000 }
gfCNCPoint1[13614] = {X 394.7459, Y 60.7909, Z -1.3333, A 0.000, B 0.000, C 0.000 }
gfCNCPoint1[13615] = {X 394.4301, Y 59.9039, Z -1.3333, A 0.000, B 0.000, C 0.000 }
gfCNCPoint1[13616] = {X 394.3179, Y 58.9691, Z -1.3333, A 0.000, B 0.000, C 0.000 }
gfCNCPoint1[13617] = {X 394.3177, Y 58.0000, Z -1.3333, A 0.000, B 0.000, C 0.000 }
gfCNCPoint1[13618] = {X 394.4240, Y 57.0565, Z -1.3333, A 0.000, B 0.000, C 0.000 }
gfCNCPoint1[13619] = {X 394.7376, Y 56.1603, Z -1.3333, A 0.000, B 0.000, C 0.000 }
gfCNCPoint1[13620] = {X 395.2428, Y 55.3564, Z -1.3333, A 0.000, B 0.000, C 0.000 }
gfCNCPoint1[13621] = {X 395.9141, Y 54.6850, Z -1.3333, A 0.000, B 0.000, C 0.000 }
gfCNCPoint1[13622] = {X 396.7181, Y 54.1799, Z -1.3333, A 0.000, B 0.000, C 0.000 }
gfCNCPoint1[13623] = {X 397.6142, Y 53.8663, Z -1.3333, A 0.000, B 0.000, C 0.000 }
gfCNCPoint1[13624] = {X 398.5577, Y 53.7600, Z -1.3333, A 0.000, B 0.000, C 0.000 }
gfCNCPoint1[13625] = {X 419.4886, Y 53.7600, Z -1.3333, A 0.000, B 0.000, C 0.000 }
gfCNCPoint1[13626] = {X 420.4321, Y 53.8663, Z -1.3333, A 0.000, B 0.000, C 0.000 }
gfCNCPoint1[13627] = {X 421.3283, Y 54.1799, Z -1.3333, A 0.000, B 0.000, C 0.000 }
gfCNCPoint1[13628] = {X 422.1322, Y 54.6850, Z -1.3333, A 0.000, B 0.000, C 0.000 }
gfCNCPoint1[13629] = {X 422.8036, Y 55.3564, Z -1.3333, A 0.000, B 0.000, C 0.000 }
gfCNCPoint1[13630] = {X 423.3087, Y 56.1603, Z -1.3333, A 0.000, B 0.000, C 0.000 }
gfCNCPoint1[13631] = {X 423.6223, Y 57.0565, Z -1.3333, A 0.000, B 0.000, C 0.000 }
gfCNCPoint1[13632] = {X 423.7286, Y 58.0000, Z -1.3333, A 0.000, B 0.000, C 0.000 }
gfCNCPoint1[13633] = {X 423.7286, Y 58.2876, Z -1.3333, A 0.000, B 0.000, C 0.000 }
gfCNCPoint1[13634] = {X 429.5823, Y 60.5692, Z -1.3333, A 0.000, B 0.000, C 0.000 }
gfCNCPoint1[13635] = {X 457.9414, Y 71.8204, Z -1.3333, A 0.000, B 0.000, C 0.000 }
gfCNCPoint1[13636] = {X 457.9414, Y 63.1423, Z -1.3333, A 0.000, B 0.000, C 0.000 }
gfCNCPoint1[13637] = {X 457.0927, Y 62.9477, Z -1.3333, A 0.000, B 0.000, C 0.000 }
gfCNCPoint1[13638] = {X 456.3017, Y 62.5839, Z -1.3333, A 0.000, B 0.000, C 0.000 }
gfCNCPoint1[13639] = {X 455.6016, Y 62.0661, Z -1.3333, A 0.000, B 0.000, C 0.000 }
gfCNCPoint1[13640] = {X 455.0221, Y 61.4163, Z -1.3333, A 0.000, B 0.000, C 0.000 }
gfCNCPoint1[13641] = {X 454.5876, Y 60.6618, Z -1.3333, A 0.000, B 0.000, C 0.000 }
gfCNCPoint1[13642] = {X 454.3163, Y 59.8344, Z -1.3333, A 0.000, B 0.000, C 0.000 }
gfCNCPoint1[13643] = {X 454.2197, Y 58.9691, Z -1.3333, A 0.000, B 0.000, C 0.000 }
gfCNCPoint1[13644] = {X 454.2196, Y 58.0000, Z -1.3333, A 0.000, B 0.000, C 0.000 }
gfCNCPoint1[13645] = {X 454.3259, Y 57.0565, Z -1.3333, A 0.000, B 0.000, C 0.000 }
gfCNCPoint1[13646] = {X 454.6395, Y 56.1603, Z -1.3333, A 0.000, B 0.000, C 0.000 }
gfCNCPoint1[13647] = {X 455.1446, Y 55.3564, Z -1.3333, A 0.000, B 0.000, C 0.000 }
gfCNCPoint1[13648] = {X 455.8160, Y 54.6850, Z -1.3333, A 0.000, B 0.000, C 0.000 }
gfCNCPoint1[13649] = {X 456.6199, Y 54.1799, Z -1.3333, A 0.000, B 0.000, C 0.000 }
gfCNCPoint1[13650] = {X 457.5161, Y 53.8663, Z -1.3333, A 0.000, B 0.000, C 0.000 }
gfCNCPoint1[13651] = {X 458.4596, Y 53.7600, Z -1.3333, A 0.000, B 0.000, C 0.000 }
gfCNCPoint1[13652] = {X 475.0000, Y 53.7600, Z -1.3333, A 0.000, B 0.000, C 0.000 }
gfCNCPoint1[13653] = {X 475.9435, Y 53.8663, Z -1.3333, A 0.000, B 0.000, C 0.000 }
gfCNCPoint1[13654] = {X 476.8397, Y 54.1799, Z -1.3333, A 0.000, B 0.000, C 0.000 }
gfCNCPoint1[13655] = {X 477.6436, Y 54.6850, Z -1.3333, A 0.000, B 0.000, C 0.000 }
gfCNCPoint1[13656] = {X 478.3150, Y 55.3564, Z -1.3333, A 0.000, B 0.000, C 0.000 }
gfCNCPoint1[13657] = {X 478.8201, Y 56.1603, Z -1.3333, A 0.000, B 0.000, C 0.000 }
gfCNCPoint1[13658] = {X 479.1337, Y 57.0565, Z -1.3333, A 0.000, B 0.000, C 0.000 }
gfCNCPoint1[13659] = {X 479.2400, Y 58.0000, Z -1.3333, A 0.000, B 0.000, C 0.000 }
gfCNCPoint1[13660] = {X 479.2400, Y 58.9342, Z -1.3333, A 0.000, B 0.000, C 0.000 }
gfCNCPoint1[13661] = {X 479.1496, Y 59.8050, Z -1.3333, A 0.000, B 0.000, C 0.000 }
gfCNCPoint1[13662] = {X 478.8822, Y 60.6387, Z -1.3333, A 0.000, B 0.000, C 0.000 }
gfCNCPoint1[13663] = {X 478.4494, Y 61.3997, Z -1.3333, A 0.000, B 0.000, C 0.000 }
gfCNCPoint1[13664] = {X 477.8694, Y 62.0556, Z -1.3333, A 0.000, B 0.000, C 0.000 }
gfCNCPoint1[13665] = {X 477.1671, Y 62.5784, Z -1.3333, A 0.000, B 0.000, C 0.000 }
gfCNCPoint1[13666] = {X 476.3724, Y 62.9458, Z -1.3333, A 0.000, B 0.000, C 0.000 }
gfCNCPoint1[13667] = {X 475.5192, Y 63.1422, Z -1.3333, A 0.000, B 0.000, C 0.000 }
gfCNCPoint1[13668] = {X 475.5196, Y 92.8335, Z -1.3333, A 0.000, B 0.000, C 0.000 }
gfCNCPoint1[13669] = {X 475.9433, Y 92.9367, Z -1.3333, A 0.000, B 0.000, C 0.000 }
gfCNCPoint1[13670] = {X 476.3605, Y 93.0633, Z -1.3333, A 0.000, B 0.000, C 0.000 }
gfCNCPoint1[13671] = {X 477.1575, Y 93.4253, Z -1.3333, A 0.000, B 0.000, C 0.000 }
gfCNCPoint1[13672] = {X 477.8625, Y 93.9441, Z -1.3333, A 0.000, B 0.000, C 0.000 }
gfCNCPoint1[13673] = {X 478.4452, Y 94.5973, Z -1.3333, A 0.000, B 0.000, C 0.000 }
gfCNCPoint1[13674] = {X 478.8803, Y 95.3569, Z -1.3333, A 0.000, B 0.000, C 0.000 }
gfCNCPoint1[13675] = {X 479.1491, Y 96.1899, Z -1.3333, A 0.000, B 0.000, C 0.000 }
gfCNCPoint1[13676] = {X 479.2400, Y 97.0605, Z -1.3333, A 0.000, B 0.000, C 0.000 }
gfCNCPoint1[13677] = {X 479.2400, Y 98.0000, Z -1.3333, A 0.000, B 0.000, C 0.000 }
gfCNCPoint1[13678] = {X 479.1337, Y 98.9435, Z -1.3333, A 0.000, B 0.000, C 0.000 }
gfCNCPoint1[13679] = {X 478.8201, Y 99.8397, Z -1.3333, A 0.000, B 0.000, C 0.000 }
gfCNCPoint1[13680] = {X 478.3150, Y 100.6436, Z -1.3333, A 0.000, B 0.000, C 0.000 }
gfCNCPoint1[13681] = {X 477.6436, Y 101.3150, Z -1.3333, A 0.000, B 0.000, C 0.000 }
gfCNCPoint1[13682] = {X 476.8397, Y 101.8201, Z -1.3333, A 0.000, B 0.000, C 0.000 }
gfCNCPoint1[13683] = {X 475.9435, Y 102.1337, Z -1.3333, A 0.000, B 0.000, C 0.000 }
gfCNCPoint1[13684] = {X 475.0000, Y 102.2400, Z -1.3333, A 0.000, B 0.000, C 0.000 }
gfCNCPoint1[13685] = {X 458.4596, Y 102.2400, Z -1.3333, A 0.000, B 0.000, C 0.000 }
gfCNCPoint1[13686] = {X 457.5161, Y 102.1337, Z -1.3333, A 0.000, B 0.000, C 0.000 }
gfCNCPoint1[13687] = {X 456.6199, Y 101.8201, Z -1.3333, A 0.000, B 0.000, C 0.000 }
gfCNCPoint1[13688] = {X 455.8160, Y 101.3150, Z -1.3333, A 0.000, B 0.000, C 0.000 }
gfCNCPoint1[13689] = {X 455.1446, Y 100.6436, Z -1.3333, A 0.000, B 0.000, C 0.000 }
gfCNCPoint1[13690] = {X 454.6395, Y 99.8397, Z -1.3333, A 0.000, B 0.000, C 0.000 }
gfCNCPoint1[13691] = {X 454.3259, Y 98.9435, Z -1.3333, A 0.000, B 0.000, C 0.000 }
gfCNCPoint1[13692] = {X 454.2196, Y 98.0000, Z -1.3333, A 0.000, B 0.000, C 0.000 }
gfCNCPoint1[13693] = {X 454.2196, Y 97.0659, Z -1.3333, A 0.000, B 0.000, C 0.000 }
gfCNCPoint1[13694] = {X 454.3099, Y 96.1957, Z -1.3333, A 0.000, B 0.000, C 0.000 }
gfCNCPoint1[13695] = {X 454.5769, Y 95.3624, Z -1.3333, A 0.000, B 0.000, C 0.000 }
gfCNCPoint1[13696] = {X 455.0092, Y 94.6018, Z -1.3333, A 0.000, B 0.000, C 0.000 }
gfCNCPoint1[13697] = {X 455.5884, Y 93.9460, Z -1.3333, A 0.000, B 0.000, C 0.000 }
gfCNCPoint1[13698] = {X 456.2899, Y 93.4231, Z -1.3333, A 0.000, B 0.000, C 0.000 }
gfCNCPoint1[13699] = {X 457.0838, Y 93.0553, Z -1.3333, A 0.000, B 0.000, C 0.000 }
gfCNCPoint1[13700] = {X 457.9363, Y 92.8584, Z -1.3333, A 0.000, B 0.000, C 0.000 }
gfCNCPoint1[13701] = {X 457.9363, Y 85.5404, Z -1.3333, A 0.000, B 0.000, C 0.000 }
gfCNCPoint1[13702] = {X 444.8488, Y 80.4101, Z -1.3333, A 0.000, B 0.000, C 0.000 }
gfCNCPoint1[13703] = {X 419.9421, Y 96.5447, Z -1.3333, A 0.000, B 0.000, C 0.000 }
gfCNCPoint1[13704] = {X 419.9467, Y 97.0648, Z -1.3333, A 0.000, B 0.000, C 0.000 }
gfCNCPoint1[13705] = {X 419.9467, Y 98.0000, Z -1.3333, A 0.000, B 0.000, C 0.000 }
gfCNCPoint1[13706] = {X 419.8404, Y 98.9435, Z -1.3333, A 0.000, B 0.000, C 0.000 }
gfCNCPoint1[13707] = {X 419.5268, Y 99.8397, Z -1.3333, A 0.000, B 0.000, C 0.000 }
gfCNCPoint1[13708] = {X 419.0217, Y 100.6436, Z -1.3333, A 0.000, B 0.000, C 0.000 }
gfCNCPoint1[13709] = {X 418.3503, Y 101.3150, Z -1.3333, A 0.000, B 0.000, C 0.000 }
gfCNCPoint1[13710] = {X 417.5464, Y 101.8201, Z -1.3333, A 0.000, B 0.000, C 0.000 }
gfCNCPoint1[13711] = {X 416.6502, Y 102.1337, Z -1.3333, A 0.000, B 0.000, C 0.000 }
gfCNCPoint1[13712] = {X 415.7067, Y 102.2400, Z -1.3333, A 0.000, B 0.000, C 0.000 }
gfCNCPoint1[13713] = {X 396.4059, Y 102.2400, Z -1.3333, A 0.000, B 0.000, C 0.000 }
gfCNCPoint1[13714] = {X 395.4625, Y 102.1337, Z -1.3333, A 0.000, B 0.000, C 0.000 }
gfCNCPoint1[13715] = {X 394.5663, Y 101.8201, Z -1.3333, A 0.000, B 0.000, C 0.000 }
gfCNCPoint1[13716] = {X 393.7624, Y 101.3150, Z -1.3333, A 0.000, B 0.000, C 0.000 }
gfCNCPoint1[13717] = {X 393.0910, Y 100.6436, Z -1.3333, A 0.000, B 0.000, C 0.000 }
gfCNCPoint1[13718] = {X 392.5858, Y 99.8397, Z -1.3333, A 0.000, B 0.000, C 0.000 }
gfCNCPoint1[13719] = {X 392.2723, Y 98.9435, Z -1.3333, A 0.000, B 0.000, C 0.000 }
gfCNCPoint1[13720] = {X 392.1659, Y 98.0000, Z -1.3333, A 0.000, B 0.000, C 0.000 }
gfCNCPoint1[13721] = {X 392.1659, Y 97.0659, Z -1.3333, A 0.000, B 0.000, C 0.000 }
gfCNCPoint1[13722] = {X 392.2718, Y 96.1245, Z -1.3333, A 0.000, B 0.000, C 0.000 }
gfCNCPoint1[13723] = {X 392.5840, Y 95.2301, Z -1.3333, A 0.000, B 0.000, C 0.000 }
gfCNCPoint1[13724] = {X 393.0870, Y 94.4274, Z -1.3333, A 0.000, B 0.000, C 0.000 }
gfCNCPoint1[13725] = {X 393.7557, Y 93.7563, Z -1.3333, A 0.000, B 0.000, C 0.000 }
gfCNCPoint1[13726] = {X 394.5567, Y 93.2505, Z -1.3333, A 0.000, B 0.000, C 0.000 }
gfCNCPoint1[13727] = {X 395.4500, Y 92.9351, Z -1.3333, A 0.000, B 0.000, C 0.000 }
gfCNCPoint1[13728] = {X 396.3910, Y 92.8260, Z -1.3333, A 0.000, B 0.000, C 0.000 }
gfCNCPoint1[13729] = {X 397.3488, Y 92.7857, Z -1.3333, A 0.000, B 0.000, C 0.000 }
gfCNCPoint1[13730] = {X 398.3032, Y 92.6951, Z -1.3333, A 0.000, B 0.000, C 0.000 }
gfCNCPoint1[13731] = {X 398.9716, Y 92.5332, Z -1.3333, A 0.000, B 0.000, C 0.000 }
gfCNCPoint1[13732] = {X 399.5871, Y 92.2261, Z -1.3333, A 0.000, B 0.000, C 0.000 }
gfCNCPoint1[13733] = {X 413.8429, Y 83.0966, Z -1.3333, A 0.000, B 0.000, C 0.000 }
gfCNCPoint1[13734] = {X 411.6857, Y 79.7281, Z -1.3333, A 0.000, B 0.000, C 0.000 }
gfCNCPoint1[13735] = {X 413.8860, Y 83.1639, Z -1.3333, A 0.000, B 0.000, C 0.000 }
gfCNCPoint1[13736] = {X 428.4062, Y 73.8650, Z -1.3333, A 0.000, B 0.000, C 0.000 }
gfCNCPoint1[13737] = {X 403.8140, Y 64.2156, Z -1.3333, A 0.000, B 0.000, C 0.000 }
gfCNCPoint1[13738] = {X 402.1005, Y 63.6483, Z -1.3333, A 0.000, B 0.000, C 0.000 }
gfCNCPoint1[13739] = {X 400.3350, Y 63.2729, Z -1.3333, A 0.000, B 0.000, C 0.000 }
gfCNCPoint1[13740] = {X 398.5388, Y 63.0940, Z -1.3333, A 0.000, B 0.000, C 0.000 }
gfCNCPoint1[13741] = {X 397.6211, Y 62.9872, Z -1.3333, A 0.000, B 0.000, C 0.000 }
gfCNCPoint1[13742] = {X 396.7495, Y 62.6805, Z -1.3333, A 0.000, B 0.000, C 0.000 }
gfCNCPoint1[13743] = {X 395.9671, Y 62.1889, Z -1.3333, A 0.000, B 0.000, C 0.000 }
gfCNCPoint1[13744] = {X 395.3125, Y 61.5368, Z -1.3333, A 0.000, B 0.000, C 0.000 }
gfCNCPoint1[13745] = {X 394.8180, Y 60.7563, Z -1.3333, A 0.000, B 0.000, C 0.000 }
gfCNCPoint1[13746] = {X 394.5081, Y 59.8858, Z -1.3333, A 0.000, B 0.000, C 0.000 }
gfCNCPoint1[13747] = {X 394.3979, Y 58.9684, Z -1.3333, A 0.000, B 0.000, C 0.000 }
gfCNCPoint1[13748] = {X 394.3977, Y 58.0000, Z -1.3333, A 0.000, B 0.000, C 0.000 }
gfCNCPoint1[13749] = {X 394.5020, Y 57.0743, Z -1.3333, A 0.000, B 0.000, C 0.000 }
gfCNCPoint1[13750] = {X 394.8097, Y 56.1950, Z -1.3333, A 0.000, B 0.000, C 0.000 }
gfCNCPoint1[13751] = {X 395.3053, Y 55.4063, Z -1.3333, A 0.000, B 0.000, C 0.000 }
gfCNCPoint1[13752] = {X 395.9640, Y 54.7476, Z -1.3333, A 0.000, B 0.000, C 0.000 }
gfCNCPoint1[13753] = {X 396.7528, Y 54.2520, Z -1.3333, A 0.000, B 0.000, C 0.000 }
gfCNCPoint1[13754] = {X 397.6320, Y 53.9443, Z -1.3333, A 0.000, B 0.000, C 0.000 }
gfCNCPoint1[13755] = {X 398.5577, Y 53.8400, Z -1.3333, A 0.000, B 0.000, C 0.000 }
gfCNCPoint1[13756] = {X 419.4886, Y 53.8400, Z -1.3333, A 0.000, B 0.000, C 0.000 }
gfCNCPoint1[13757] = {X 420.4143, Y 53.9443, Z -1.3333, A 0.000, B 0.000, C 0.000 }
gfCNCPoint1[13758] = {X 421.2936, Y 54.2520, Z -1.3333, A 0.000, B 0.000, C 0.000 }
gfCNCPoint1[13759] = {X 422.0823, Y 54.7476, Z -1.3333, A 0.000, B 0.000, C 0.000 }
gfCNCPoint1[13760] = {X 422.7410, Y 55.4063, Z -1.3333, A 0.000, B 0.000, C 0.000 }
gfCNCPoint1[13761] = {X 423.2366, Y 56.1950, Z -1.3333, A 0.000, B 0.000, C 0.000 }
gfCNCPoint1[13762] = {X 423.5443, Y 57.0743, Z -1.3333, A 0.000, B 0.000, C 0.000 }
gfCNCPoint1[13763] = {X 423.6486, Y 58.0000, Z -1.3333, A 0.000, B 0.000, C 0.000 }
gfCNCPoint1[13764] = {X 423.6486, Y 58.3423, Z -1.3333, A 0.000, B 0.000, C 0.000 }
gfCNCPoint1[13765] = {X 429.5531, Y 60.6436, Z -1.3333, A 0.000, B 0.000, C 0.000 }
gfCNCPoint1[13766] = {X 458.0214, Y 71.9382, Z -1.3333, A 0.000, B 0.000, C 0.000 }
gfCNCPoint1[13767] = {X 458.0214, Y 63.0709, Z -1.3333, A 0.000, B 0.000, C 0.000 }
gfCNCPoint1[13768] = {X 457.9191, Y 63.0588, Z -1.3333, A 0.000, B 0.000, C 0.000 }
gfCNCPoint1[13769] = {X 457.8172, Y 63.0442, Z -1.3333, A 0.000, B 0.000, C 0.000 }
gfCNCPoint1[13770] = {X 456.8794, Y 62.7823, Z -1.3333, A 0.000, B 0.000, C 0.000 }
gfCNCPoint1[13771] = {X 456.0282, Y 62.3096, Z -1.3333, A 0.000, B 0.000, C 0.000 }
gfCNCPoint1[13772] = {X 455.3102, Y 61.6520, Z -1.3333, A 0.000, B 0.000, C 0.000 }
gfCNCPoint1[13773] = {X 454.7648, Y 60.8455, Z -1.3333, A 0.000, B 0.000, C 0.000 }
gfCNCPoint1[13774] = {X 454.4217, Y 59.9344, Z -1.3333, A 0.000, B 0.000, C 0.000 }
gfCNCPoint1[13775] = {X 454.2997, Y 58.9684, Z -1.3333, A 0.000, B 0.000, C 0.000 }
gfCNCPoint1[13776] = {X 454.2996, Y 58.0000, Z -1.3333, A 0.000, B 0.000, C 0.000 }
gfCNCPoint1[13777] = {X 454.4039, Y 57.0743, Z -1.3333, A 0.000, B 0.000, C 0.000 }
gfCNCPoint1[13778] = {X 454.7116, Y 56.1950, Z -1.3333, A 0.000, B 0.000, C 0.000 }
gfCNCPoint1[13779] = {X 455.2072, Y 55.4063, Z -1.3333, A 0.000, B 0.000, C 0.000 }
gfCNCPoint1[13780] = {X 455.8659, Y 54.7476, Z -1.3333, A 0.000, B 0.000, C 0.000 }
gfCNCPoint1[13781] = {X 456.6546, Y 54.2520, Z -1.3333, A 0.000, B 0.000, C 0.000 }
gfCNCPoint1[13782] = {X 457.5339, Y 53.9443, Z -1.3333, A 0.000, B 0.000, C 0.000 }
gfCNCPoint1[13783] = {X 458.4596, Y 53.8400, Z -1.3333, A 0.000, B 0.000, C 0.000 }
gfCNCPoint1[13784] = {X 475.0000, Y 53.8400, Z -1.3333, A 0.000, B 0.000, C 0.000 }
gfCNCPoint1[13785] = {X 475.9257, Y 53.9443, Z -1.3333, A 0.000, B 0.000, C 0.000 }
gfCNCPoint1[13786] = {X 476.8050, Y 54.2520, Z -1.3333, A 0.000, B 0.000, C 0.000 }
gfCNCPoint1[13787] = {X 477.5937, Y 54.7476, Z -1.3333, A 0.000, B 0.000, C 0.000 }
gfCNCPoint1[13788] = {X 478.2524, Y 55.4063, Z -1.3333, A 0.000, B 0.000, C 0.000 }
gfCNCPoint1[13789] = {X 478.7480, Y 56.1950, Z -1.3333, A 0.000, B 0.000, C 0.000 }
gfCNCPoint1[13790] = {X 479.0557, Y 57.0743, Z -1.3333, A 0.000, B 0.000, C 0.000 }
gfCNCPoint1[13791] = {X 479.1600, Y 58.0000, Z -1.3333, A 0.000, B 0.000, C 0.000 }
gfCNCPoint1[13792] = {X 479.1600, Y 58.9342, Z -1.3333, A 0.000, B 0.000, C 0.000 }
gfCNCPoint1[13793] = {X 479.0692, Y 59.7985, Z -1.3333, A 0.000, B 0.000, C 0.000 }
gfCNCPoint1[13794] = {X 478.8008, Y 60.6250, Z -1.3333, A 0.000, B 0.000, C 0.000 }
gfCNCPoint1[13795] = {X 478.3666, Y 61.3778, Z -1.3333, A 0.000, B 0.000, C 0.000 }
gfCNCPoint1[13796] = {X 477.7854, Y 62.0239, Z -1.3333, A 0.000, B 0.000, C 0.000 }
gfCNCPoint1[13797] = {X 477.0827, Y 62.5352, Z -1.3333, A 0.000, B 0.000, C 0.000 }
gfCNCPoint1[13798] = {X 476.2891, Y 62.8893, Z -1.3333, A 0.000, B 0.000, C 0.000 }
gfCNCPoint1[13799] = {X 475.4392, Y 63.0708, Z -1.3333, A 0.000, B 0.000, C 0.000 }
gfCNCPoint1[13800] = {X 475.4396, Y 92.8984, Z -1.3333, A 0.000, B 0.000, C 0.000 }
gfCNCPoint1[13801] = {X 475.8910, Y 93.0054, Z -1.3333, A 0.000, B 0.000, C 0.000 }
gfCNCPoint1[13802] = {X 476.3352, Y 93.1392, Z -1.3333, A 0.000, B 0.000, C 0.000 }
gfCNCPoint1[13803] = {X 477.1170, Y 93.4943, Z -1.3333, A 0.000, B 0.000, C 0.000 }
gfCNCPoint1[13804] = {X 477.8087, Y 94.0032, Z -1.3333, A 0.000, B 0.000, C 0.000 }
gfCNCPoint1[13805] = {X 478.3803, Y 94.6441, Z -1.3333, A 0.000, B 0.000, C 0.000 }
gfCNCPoint1[13806] = {X 478.8071, Y 95.3892, Z -1.3333, A 0.000, B 0.000, C 0.000 }
gfCNCPoint1[13807] = {X 479.0708, Y 96.2065, Z -1.3333, A 0.000, B 0.000, C 0.000 }
gfCNCPoint1[13808] = {X 479.1600, Y 97.0605, Z -1.3333, A 0.000, B 0.000, C 0.000 }
gfCNCPoint1[13809] = {X 479.1600, Y 98.0000, Z -1.3333, A 0.000, B 0.000, C 0.000 }
gfCNCPoint1[13810] = {X 479.0557, Y 98.9257, Z -1.3333, A 0.000, B 0.000, C 0.000 }
gfCNCPoint1[13811] = {X 478.7480, Y 99.8050, Z -1.3333, A 0.000, B 0.000, C 0.000 }
gfCNCPoint1[13812] = {X 478.2524, Y 100.5937, Z -1.3333, A 0.000, B 0.000, C 0.000 }
gfCNCPoint1[13813] = {X 477.5937, Y 101.2524, Z -1.3333, A 0.000, B 0.000, C 0.000 }
gfCNCPoint1[13814] = {X 476.8050, Y 101.7480, Z -1.3333, A 0.000, B 0.000, C 0.000 }
gfCNCPoint1[13815] = {X 475.9257, Y 102.0557, Z -1.3333, A 0.000, B 0.000, C 0.000 }
gfCNCPoint1[13816] = {X 475.0000, Y 102.1600, Z -1.3333, A 0.000, B 0.000, C 0.000 }
gfCNCPoint1[13817] = {X 458.4596, Y 102.1600, Z -1.3333, A 0.000, B 0.000, C 0.000 }
gfCNCPoint1[13818] = {X 457.5339, Y 102.0557, Z -1.3333, A 0.000, B 0.000, C 0.000 }
gfCNCPoint1[13819] = {X 456.6546, Y 101.7480, Z -1.3333, A 0.000, B 0.000, C 0.000 }
gfCNCPoint1[13820] = {X 455.8659, Y 101.2524, Z -1.3333, A 0.000, B 0.000, C 0.000 }
gfCNCPoint1[13821] = {X 455.2072, Y 100.5937, Z -1.3333, A 0.000, B 0.000, C 0.000 }
gfCNCPoint1[13822] = {X 454.7116, Y 99.8050, Z -1.3333, A 0.000, B 0.000, C 0.000 }
gfCNCPoint1[13823] = {X 454.4039, Y 98.9257, Z -1.3333, A 0.000, B 0.000, C 0.000 }
gfCNCPoint1[13824] = {X 454.2996, Y 98.0000, Z -1.3333, A 0.000, B 0.000, C 0.000 }
gfCNCPoint1[13825] = {X 454.2996, Y 97.0659, Z -1.3333, A 0.000, B 0.000, C 0.000 }
gfCNCPoint1[13826] = {X 454.3903, Y 96.2022, Z -1.3333, A 0.000, B 0.000, C 0.000 }
gfCNCPoint1[13827] = {X 454.6583, Y 95.3761, Z -1.3333, A 0.000, B 0.000, C 0.000 }
gfCNCPoint1[13828] = {X 455.0920, Y 94.6237, Z -1.3333, A 0.000, B 0.000, C 0.000 }
gfCNCPoint1[13829] = {X 455.6724, Y 93.9777, Z -1.3333, A 0.000, B 0.000, C 0.000 }
gfCNCPoint1[13830] = {X 456.3743, Y 93.4663, Z -1.3333, A 0.000, B 0.000, C 0.000 }
gfCNCPoint1[13831] = {X 457.1672, Y 93.1118, Z -1.3333, A 0.000, B 0.000, C 0.000 }
gfCNCPoint1[13832] = {X 458.0163, Y 92.9296, Z -1.3333, A 0.000, B 0.000, C 0.000 }
gfCNCPoint1[13833] = {X 458.0163, Y 85.4858, Z -1.3333, A 0.000, B 0.000, C 0.000 }
gfCNCPoint1[13834] = {X 444.8398, Y 80.3206, Z -1.3333, A 0.000, B 0.000, C 0.000 }
gfCNCPoint1[13835] = {X 419.8617, Y 96.5015, Z -1.3333, A 0.000, B 0.000, C 0.000 }
gfCNCPoint1[13836] = {X 419.8667, Y 97.0652, Z -1.3333, A 0.000, B 0.000, C 0.000 }
gfCNCPoint1[13837] = {X 419.8667, Y 98.0000, Z -1.3333, A 0.000, B 0.000, C 0.000 }
gfCNCPoint1[13838] = {X 419.7624, Y 98.9257, Z -1.3333, A 0.000, B 0.000, C 0.000 }
gfCNCPoint1[13839] = {X 419.4547, Y 99.8050, Z -1.3333, A 0.000, B 0.000, C 0.000 }
gfCNCPoint1[13840] = {X 418.9591, Y 100.5937, Z -1.3333, A 0.000, B 0.000, C 0.000 }
gfCNCPoint1[13841] = {X 418.3004, Y 101.2524, Z -1.3333, A 0.000, B 0.000, C 0.000 }
gfCNCPoint1[13842] = {X 417.5117, Y 101.7480, Z -1.3333, A 0.000, B 0.000, C 0.000 }
gfCNCPoint1[13843] = {X 416.6324, Y 102.0557, Z -1.3333, A 0.000, B 0.000, C 0.000 }
gfCNCPoint1[13844] = {X 415.7067, Y 102.1600, Z -1.3333, A 0.000, B 0.000, C 0.000 }
gfCNCPoint1[13845] = {X 396.4059, Y 102.1600, Z -1.3333, A 0.000, B 0.000, C 0.000 }
gfCNCPoint1[13846] = {X 395.4803, Y 102.0557, Z -1.3333, A 0.000, B 0.000, C 0.000 }
gfCNCPoint1[13847] = {X 394.6010, Y 101.7480, Z -1.3333, A 0.000, B 0.000, C 0.000 }
gfCNCPoint1[13848] = {X 393.8122, Y 101.2524, Z -1.3333, A 0.000, B 0.000, C 0.000 }
gfCNCPoint1[13849] = {X 393.1535, Y 100.5937, Z -1.3333, A 0.000, B 0.000, C 0.000 }
gfCNCPoint1[13850] = {X 392.6579, Y 99.8050, Z -1.3333, A 0.000, B 0.000, C 0.000 }
gfCNCPoint1[13851] = {X 392.3502, Y 98.9257, Z -1.3333, A 0.000, B 0.000, C 0.000 }
gfCNCPoint1[13852] = {X 392.2459, Y 98.0000, Z -1.3333, A 0.000, B 0.000, C 0.000 }
gfCNCPoint1[13853] = {X 392.2459, Y 97.0659, Z -1.3333, A 0.000, B 0.000, C 0.000 }
gfCNCPoint1[13854] = {X 392.3498, Y 96.1422, Z -1.3333, A 0.000, B 0.000, C 0.000 }
gfCNCPoint1[13855] = {X 392.6562, Y 95.2646, Z -1.3333, A 0.000, B 0.000, C 0.000 }
gfCNCPoint1[13856] = {X 393.1497, Y 94.4770, Z -1.3333, A 0.000, B 0.000, C 0.000 }
gfCNCPoint1[13857] = {X 393.8059, Y 93.8186, Z -1.3333, A 0.000, B 0.000, C 0.000 }
gfCNCPoint1[13858] = {X 394.5919, Y 93.3223, Z -1.3333, A 0.000, B 0.000, C 0.000 }
gfCNCPoint1[13859] = {X 395.4684, Y 93.0130, Z -1.3333, A 0.000, B 0.000, C 0.000 }
gfCNCPoint1[13860] = {X 396.3918, Y 92.9060, Z -1.3333, A 0.000, B 0.000, C 0.000 }
gfCNCPoint1[13861] = {X 397.3541, Y 92.8655, Z -1.3333, A 0.000, B 0.000, C 0.000 }
gfCNCPoint1[13862] = {X 398.3130, Y 92.7745, Z -1.3333, A 0.000, B 0.000, C 0.000 }
gfCNCPoint1[13863] = {X 398.9990, Y 92.6083, Z -1.3333, A 0.000, B 0.000, C 0.000 }
gfCNCPoint1[13864] = {X 399.6306, Y 92.2933, Z -1.3333, A 0.000, B 0.000, C 0.000 }
gfCNCPoint1[13865] = {X 413.8860, Y 83.1639, Z -1.3333, A 0.000, B 0.000, C 0.000 }
gfCNCPoint1[13866] = {X 411.7288, Y 79.7955, Z -1.3333, A 0.000, B 0.000, C 0.000 }
gfCNCPoint1[13867] = {X 413.9292, Y 83.2313, Z -1.3333, A 0.000, B 0.000, C 0.000 }
gfCNCPoint1[13868] = {X 428.5814, Y 73.8478, Z -1.3333, A 0.000, B 0.000, C 0.000 }
gfCNCPoint1[13869] = {X 403.8433, Y 64.1412, Z -1.3333, A 0.000, B 0.000, C 0.000 }
gfCNCPoint1[13870] = {X 402.1209, Y 63.5709, Z -1.3333, A 0.000, B 0.000, C 0.000 }
gfCNCPoint1[13871] = {X 400.3462, Y 63.1937, Z -1.3333, A 0.000, B 0.000, C 0.000 }
gfCNCPoint1[13872] = {X 398.5408, Y 63.0140, Z -1.3333, A 0.000, B 0.000, C 0.000 }
gfCNCPoint1[13873] = {X 397.6404, Y 62.9096, Z -1.3333, A 0.000, B 0.000, C 0.000 }
gfCNCPoint1[13874] = {X 396.7853, Y 62.6089, Z -1.3333, A 0.000, B 0.000, C 0.000 }
gfCNCPoint1[13875] = {X 396.0176, Y 62.1269, Z -1.3333, A 0.000, B 0.000, C 0.000 }
gfCNCPoint1[13876] = {X 395.3753, Y 61.4873, Z -1.3333, A 0.000, B 0.000, C 0.000 }
gfCNCPoint1[13877] = {X 394.8902, Y 60.7216, Z -1.3333, A 0.000, B 0.000, C 0.000 }
gfCNCPoint1[13878] = {X 394.5860, Y 59.8677, Z -1.3333, A 0.000, B 0.000, C 0.000 }
gfCNCPoint1[13879] = {X 394.4779, Y 58.9678, Z -1.3333, A 0.000, B 0.000, C 0.000 }
gfCNCPoint1[13880] = {X 394.4777, Y 58.0000, Z -1.3333, A 0.000, B 0.000, C 0.000 }
gfCNCPoint1[13881] = {X 394.5800, Y 57.0921, Z -1.3333, A 0.000, B 0.000, C 0.000 }
gfCNCPoint1[13882] = {X 394.8818, Y 56.2298, Z -1.3333, A 0.000, B 0.000, C 0.000 }
gfCNCPoint1[13883] = {X 395.3679, Y 55.4562, Z -1.3333, A 0.000, B 0.000, C 0.000 }
gfCNCPoint1[13884] = {X 396.0139, Y 54.8101, Z -1.3333, A 0.000, B 0.000, C 0.000 }
gfCNCPoint1[13885] = {X 396.7875, Y 54.3240, Z -1.3333, A 0.000, B 0.000, C 0.000 }
gfCNCPoint1[13886] = {X 397.6498, Y 54.0223, Z -1.3333, A 0.000, B 0.000, C 0.000 }
gfCNCPoint1[13887] = {X 398.5577, Y 53.9200, Z -1.3333, A 0.000, B 0.000, C 0.000 }
gfCNCPoint1[13888] = {X 419.4886, Y 53.9200, Z -1.3333, A 0.000, B 0.000, C 0.000 }
gfCNCPoint1[13889] = {X 420.3965, Y 54.0223, Z -1.3333, A 0.000, B 0.000, C 0.000 }
gfCNCPoint1[13890] = {X 421.2589, Y 54.3240, Z -1.3333, A 0.000, B 0.000, C 0.000 }
gfCNCPoint1[13891] = {X 422.0324, Y 54.8101, Z -1.3333, A 0.000, B 0.000, C 0.000 }
gfCNCPoint1[13892] = {X 422.6785, Y 55.4562, Z -1.3333, A 0.000, B 0.000, C 0.000 }
gfCNCPoint1[13893] = {X 423.1646, Y 56.2298, Z -1.3333, A 0.000, B 0.000, C 0.000 }
gfCNCPoint1[13894] = {X 423.4663, Y 57.0921, Z -1.3333, A 0.000, B 0.000, C 0.000 }
gfCNCPoint1[13895] = {X 423.5686, Y 58.0000, Z -1.3333, A 0.000, B 0.000, C 0.000 }
gfCNCPoint1[13896] = {X 423.5686, Y 58.3970, Z -1.3333, A 0.000, B 0.000, C 0.000 }
gfCNCPoint1[13897] = {X 429.5238, Y 60.7181, Z -1.3333, A 0.000, B 0.000, C 0.000 }
gfCNCPoint1[13898] = {X 458.1014, Y 72.0560, Z -1.3333, A 0.000, B 0.000, C 0.000 }
gfCNCPoint1[13899] = {X 458.1014, Y 62.9983, Z -1.3333, A 0.000, B 0.000, C 0.000 }
gfCNCPoint1[13900] = {X 457.9652, Y 62.9840, Z -1.3333, A 0.000, B 0.000, C 0.000 }
gfCNCPoint1[13901] = {X 457.8295, Y 62.9651, Z -1.3333, A 0.000, B 0.000, C 0.000 }
gfCNCPoint1[13902] = {X 456.9098, Y 62.7083, Z -1.3333, A 0.000, B 0.000, C 0.000 }
gfCNCPoint1[13903] = {X 456.0750, Y 62.2447, Z -1.3333, A 0.000, B 0.000, C 0.000 }
gfCNCPoint1[13904] = {X 455.3708, Y 61.5997, Z -1.3333, A 0.000, B 0.000, C 0.000 }
gfCNCPoint1[13905] = {X 454.8358, Y 60.8088, Z -1.3333, A 0.000, B 0.000, C 0.000 }
gfCNCPoint1[13906] = {X 454.4993, Y 59.9151, Z -1.3333, A 0.000, B 0.000, C 0.000 }
gfCNCPoint1[13907] = {X 454.3797, Y 58.9678, Z -1.3333, A 0.000, B 0.000, C 0.000 }
gfCNCPoint1[13908] = {X 454.3796, Y 58.0000, Z -1.3333, A 0.000, B 0.000, C 0.000 }
gfCNCPoint1[13909] = {X 454.4819, Y 57.0921, Z -1.3333, A 0.000, B 0.000, C 0.000 }
gfCNCPoint1[13910] = {X 454.7837, Y 56.2298, Z -1.3333, A 0.000, B 0.000, C 0.000 }
gfCNCPoint1[13911] = {X 455.2697, Y 55.4562, Z -1.3333, A 0.000, B 0.000, C 0.000 }
gfCNCPoint1[13912] = {X 455.9158, Y 54.8101, Z -1.3333, A 0.000, B 0.000, C 0.000 }
gfCNCPoint1[13913] = {X 456.6894, Y 54.3240, Z -1.3333, A 0.000, B 0.000, C 0.000 }
gfCNCPoint1[13914] = {X 457.5517, Y 54.0223, Z -1.3333, A 0.000, B 0.000, C 0.000 }
gfCNCPoint1[13915] = {X 458.4596, Y 53.9200, Z -1.3333, A 0.000, B 0.000, C 0.000 }
gfCNCPoint1[13916] = {X 475.0000, Y 53.9200, Z -1.3333, A 0.000, B 0.000, C 0.000 }
gfCNCPoint1[13917] = {X 475.9079, Y 54.0223, Z -1.3333, A 0.000, B 0.000, C 0.000 }
gfCNCPoint1[13918] = {X 476.7702, Y 54.3240, Z -1.3333, A 0.000, B 0.000, C 0.000 }
gfCNCPoint1[13919] = {X 477.5438, Y 54.8101, Z -1.3333, A 0.000, B 0.000, C 0.000 }
gfCNCPoint1[13920] = {X 478.1899, Y 55.4562, Z -1.3333, A 0.000, B 0.000, C 0.000 }
gfCNCPoint1[13921] = {X 478.6760, Y 56.2298, Z -1.3333, A 0.000, B 0.000, C 0.000 }
gfCNCPoint1[13922] = {X 478.9777, Y 57.0921, Z -1.3333, A 0.000, B 0.000, C 0.000 }
gfCNCPoint1[13923] = {X 479.0800, Y 58.0000, Z -1.3333, A 0.000, B 0.000, C 0.000 }
gfCNCPoint1[13924] = {X 479.0800, Y 58.9342, Z -1.3333, A 0.000, B 0.000, C 0.000 }
gfCNCPoint1[13925] = {X 478.9888, Y 59.7919, Z -1.3333, A 0.000, B 0.000, C 0.000 }
gfCNCPoint1[13926] = {X 478.7193, Y 60.6113, Z -1.3333, A 0.000, B 0.000, C 0.000 }
gfCNCPoint1[13927] = {X 478.2836, Y 61.3557, Z -1.3333, A 0.000, B 0.000, C 0.000 }
gfCNCPoint1[13928] = {X 477.7012, Y 61.9918, Z -1.3333, A 0.000, B 0.000, C 0.000 }
gfCNCPoint1[13929] = {X 476.9980, Y 62.4914, Z -1.3333, A 0.000, B 0.000, C 0.000 }
gfCNCPoint1[13930] = {X 476.2056, Y 62.8319, Z -1.3333, A 0.000, B 0.000, C 0.000 }
gfCNCPoint1[13931] = {X 475.3592, Y 62.9982, Z -1.3333, A 0.000, B 0.000, C 0.000 }
gfCNCPoint1[13932] = {X 475.3596, Y 92.9639, Z -1.3333, A 0.000, B 0.000, C 0.000 }
gfCNCPoint1[13933] = {X 475.8387, Y 93.0743, Z -1.3333, A 0.000, B 0.000, C 0.000 }
gfCNCPoint1[13934] = {X 476.3098, Y 93.2150, Z -1.3333, A 0.000, B 0.000, C 0.000 }
gfCNCPoint1[13935] = {X 477.0766, Y 93.5633, Z -1.3333, A 0.000, B 0.000, C 0.000 }
gfCNCPoint1[13936] = {X 477.7548, Y 94.0624, Z -1.3333, A 0.000, B 0.000, C 0.000 }
gfCNCPoint1[13937] = {X 478.3154, Y 94.6909, Z -1.3333, A 0.000, B 0.000, C 0.000 }
gfCNCPoint1[13938] = {X 478.7339, Y 95.4216, Z -1.3333, A 0.000, B 0.000, C 0.000 }
gfCNCPoint1[13939] = {X 478.9925, Y 96.2230, Z -1.3333, A 0.000, B 0.000, C 0.000 }
gfCNCPoint1[13940] = {X 479.0800, Y 97.0605, Z -1.3333, A 0.000, B 0.000, C 0.000 }
gfCNCPoint1[13941] = {X 479.0800, Y 98.0000, Z -1.3333, A 0.000, B 0.000, C 0.000 }
gfCNCPoint1[13942] = {X 478.9777, Y 98.9079, Z -1.3333, A 0.000, B 0.000, C 0.000 }
gfCNCPoint1[13943] = {X 478.6760, Y 99.7702, Z -1.3333, A 0.000, B 0.000, C 0.000 }
gfCNCPoint1[13944] = {X 478.1899, Y 100.5438, Z -1.3333, A 0.000, B 0.000, C 0.000 }
gfCNCPoint1[13945] = {X 477.5438, Y 101.1899, Z -1.3333, A 0.000, B 0.000, C 0.000 }
gfCNCPoint1[13946] = {X 476.7702, Y 101.6760, Z -1.3333, A 0.000, B 0.000, C 0.000 }
gfCNCPoint1[13947] = {X 475.9079, Y 101.9777, Z -1.3333, A 0.000, B 0.000, C 0.000 }
gfCNCPoint1[13948] = {X 475.0000, Y 102.0800, Z -1.3333, A 0.000, B 0.000, C 0.000 }
gfCNCPoint1[13949] = {X 458.4596, Y 102.0800, Z -1.3333, A 0.000, B 0.000, C 0.000 }
gfCNCPoint1[13950] = {X 457.5517, Y 101.9777, Z -1.3333, A 0.000, B 0.000, C 0.000 }
gfCNCPoint1[13951] = {X 456.6894, Y 101.6760, Z -1.3333, A 0.000, B 0.000, C 0.000 }
gfCNCPoint1[13952] = {X 455.9158, Y 101.1899, Z -1.3333, A 0.000, B 0.000, C 0.000 }
gfCNCPoint1[13953] = {X 455.2697, Y 100.5438, Z -1.3333, A 0.000, B 0.000, C 0.000 }
gfCNCPoint1[13954] = {X 454.7837, Y 99.7702, Z -1.3333, A 0.000, B 0.000, C 0.000 }
gfCNCPoint1[13955] = {X 454.4819, Y 98.9079, Z -1.3333, A 0.000, B 0.000, C 0.000 }
gfCNCPoint1[13956] = {X 454.3796, Y 98.0000, Z -1.3333, A 0.000, B 0.000, C 0.000 }
gfCNCPoint1[13957] = {X 454.3796, Y 97.0659, Z -1.3333, A 0.000, B 0.000, C 0.000 }
gfCNCPoint1[13958] = {X 454.4707, Y 96.2088, Z -1.3333, A 0.000, B 0.000, C 0.000 }
gfCNCPoint1[13959] = {X 454.7398, Y 95.3899, Z -1.3333, A 0.000, B 0.000, C 0.000 }
gfCNCPoint1[13960] = {X 455.1749, Y 94.6458, Z -1.3333, A 0.000, B 0.000, C 0.000 }
gfCNCPoint1[13961] = {X 455.7566, Y 94.0098, Z -1.3333, A 0.000, B 0.000, C 0.000 }
gfCNCPoint1[13962] = {X 456.4590, Y 93.5101, Z -1.3333, A 0.000, B 0.000, C 0.000 }
gfCNCPoint1[13963] = {X 457.2507, Y 93.1692, Z -1.3333, A 0.000, B 0.000, C 0.000 }
gfCNCPoint1[13964] = {X 458.0963, Y 93.0021, Z -1.3333, A 0.000, B 0.000, C 0.000 }
gfCNCPoint1[13965] = {X 458.0963, Y 85.4313, Z -1.3333, A 0.000, B 0.000, C 0.000 }
gfCNCPoint1[13966] = {X 444.8307, Y 80.2311, Z -1.3333, A 0.000, B 0.000, C 0.000 }
gfCNCPoint1[13967] = {X 419.7813, Y 96.4582, Z -1.3333, A 0.000, B 0.000, C 0.000 }
gfCNCPoint1[13968] = {X 419.7867, Y 97.0656, Z -1.3333, A 0.000, B 0.000, C 0.000 }
gfCNCPoint1[13969] = {X 419.7867, Y 98.0000, Z -1.3333, A 0.000, B 0.000, C 0.000 }
gfCNCPoint1[13970] = {X 419.6844, Y 98.9079, Z -1.3333, A 0.000, B 0.000, C 0.000 }
gfCNCPoint1[13971] = {X 419.3827, Y 99.7702, Z -1.3333, A 0.000, B 0.000, C 0.000 }
gfCNCPoint1[13972] = {X 418.8966, Y 100.5438, Z -1.3333, A 0.000, B 0.000, C 0.000 }
gfCNCPoint1[13973] = {X 418.2505, Y 101.1899, Z -1.3333, A 0.000, B 0.000, C 0.000 }
gfCNCPoint1[13974] = {X 417.4769, Y 101.6760, Z -1.3333, A 0.000, B 0.000, C 0.000 }
gfCNCPoint1[13975] = {X 416.6146, Y 101.9777, Z -1.3333, A 0.000, B 0.000, C 0.000 }
gfCNCPoint1[13976] = {X 415.7067, Y 102.0800, Z -1.3333, A 0.000, B 0.000, C 0.000 }
gfCNCPoint1[13977] = {X 396.4059, Y 102.0800, Z -1.3333, A 0.000, B 0.000, C 0.000 }
gfCNCPoint1[13978] = {X 395.4981, Y 101.9777, Z -1.3333, A 0.000, B 0.000, C 0.000 }
gfCNCPoint1[13979] = {X 394.6357, Y 101.6760, Z -1.3333, A 0.000, B 0.000, C 0.000 }
gfCNCPoint1[13980] = {X 393.8621, Y 101.1899, Z -1.3333, A 0.000, B 0.000, C 0.000 }
gfCNCPoint1[13981] = {X 393.2161, Y 100.5438, Z -1.3333, A 0.000, B 0.000, C 0.000 }
gfCNCPoint1[13982] = {X 392.7300, Y 99.7702, Z -1.3333, A 0.000, B 0.000, C 0.000 }
gfCNCPoint1[13983] = {X 392.4282, Y 98.9079, Z -1.3333, A 0.000, B 0.000, C 0.000 }
gfCNCPoint1[13984] = {X 392.3259, Y 98.0000, Z -1.3333, A 0.000, B 0.000, C 0.000 }
gfCNCPoint1[13985] = {X 392.3259, Y 97.0659, Z -1.3333, A 0.000, B 0.000, C 0.000 }
gfCNCPoint1[13986] = {X 392.4278, Y 96.1599, Z -1.3333, A 0.000, B 0.000, C 0.000 }
gfCNCPoint1[13987] = {X 392.7283, Y 95.2991, Z -1.3333, A 0.000, B 0.000, C 0.000 }
gfCNCPoint1[13988] = {X 393.2125, Y 94.5266, Z -1.3333, A 0.000, B 0.000, C 0.000 }
gfCNCPoint1[13989] = {X 393.8561, Y 93.8808, Z -1.3333, A 0.000, B 0.000, C 0.000 }
gfCNCPoint1[13990] = {X 394.6271, Y 93.3941, Z -1.3333, A 0.000, B 0.000, C 0.000 }
gfCNCPoint1[13991] = {X 395.4869, Y 93.0908, Z -1.3333, A 0.000, B 0.000, C 0.000 }
gfCNCPoint1[13992] = {X 396.3925, Y 92.9860, Z -1.3333, A 0.000, B 0.000, C 0.000 }
gfCNCPoint1[13993] = {X 397.3594, Y 92.9453, Z -1.3333, A 0.000, B 0.000, C 0.000 }
gfCNCPoint1[13994] = {X 398.3228, Y 92.8538, Z -1.3333, A 0.000, B 0.000, C 0.000 }
gfCNCPoint1[13995] = {X 399.0264, Y 92.6835, Z -1.3333, A 0.000, B 0.000, C 0.000 }
gfCNCPoint1[13996] = {X 399.6742, Y 92.3604, Z -1.3333, A 0.000, B 0.000, C 0.000 }
gfCNCPoint1[13997] = {X 413.9292, Y 83.2313, Z -1.3333, A 0.000, B 0.000, C 0.000 }
gfCNCPoint1[13998] = {X 411.7654, Y 79.8526, Z -1.3333, A 0.000, B 0.000, C 0.000 }
gfCNCPoint1[13999] = {X 411.7678, Y 79.8511, Z -1.3333, A 0.000, B 0.000, C 0.000 }
gfCNCPoint1[14000] = {X 413.9657, Y 83.2885, Z -1.3333, A 0.000, B 0.000, C 0.000 }
gfCNCPoint1[14001] = {X 428.7567, Y 73.8306, Z -1.3333, A 0.000, B 0.000, C 0.000 }
gfCNCPoint1[14002] = {X 403.8726, Y 64.0667, Z -1.3333, A 0.000, B 0.000, C 0.000 }
gfCNCPoint1[14003] = {X 402.1413, Y 63.4936, Z -1.3333, A 0.000, B 0.000, C 0.000 }
gfCNCPoint1[14004] = {X 400.3575, Y 63.1145, Z -1.3333, A 0.000, B 0.000, C 0.000 }
gfCNCPoint1[14005] = {X 398.5427, Y 62.9340, Z -1.3333, A 0.000, B 0.000, C 0.000 }
gfCNCPoint1[14006] = {X 397.6551, Y 62.8309, Z -1.3333, A 0.000, B 0.000, C 0.000 }
gfCNCPoint1[14007] = {X 396.8125, Y 62.5333, Z -1.3333, A 0.000, B 0.000, C 0.000 }
gfCNCPoint1[14008] = {X 396.0571, Y 62.0560, Z -1.3333, A 0.000, B 0.000, C 0.000 }
gfCNCPoint1[14009] = {X 395.4264, Y 61.4230, Z -1.3333, A 0.000, B 0.000, C 0.000 }
gfCNCPoint1[14010] = {X 394.9520, Y 60.6657, Z -1.3333, A 0.000, B 0.000, C 0.000 }
gfCNCPoint1[14011] = {X 394.6575, Y 59.8220, Z -1.3333, A 0.000, B 0.000, C 0.000 }
gfCNCPoint1[14012] = {X 394.5577, Y 58.9340, Z -1.3333, A 0.000, B 0.000, C 0.000 }
gfCNCPoint1[14013] = {X 394.5577, Y 58.0000, Z -1.3333, A 0.000, B 0.000, C 0.000 }
gfCNCPoint1[14014] = {X 394.6580, Y 57.1099, Z -1.3333, A 0.000, B 0.000, C 0.000 }
gfCNCPoint1[14015] = {X 394.9538, Y 56.2645, Z -1.3333, A 0.000, B 0.000, C 0.000 }
gfCNCPoint1[14016] = {X 395.4304, Y 55.5060, Z -1.3333, A 0.000, B 0.000, C 0.000 }
gfCNCPoint1[14017] = {X 396.0638, Y 54.8727, Z -1.3333, A 0.000, B 0.000, C 0.000 }
gfCNCPoint1[14018] = {X 396.8222, Y 54.3961, Z -1.3333, A 0.000, B 0.000, C 0.000 }
gfCNCPoint1[14019] = {X 397.6676, Y 54.1003, Z -1.3333, A 0.000, B 0.000, C 0.000 }
gfCNCPoint1[14020] = {X 398.5577, Y 54.0000, Z -1.3333, A 0.000, B 0.000, C 0.000 }
gfCNCPoint1[14021] = {X 419.4886, Y 54.0000, Z -1.3333, A 0.000, B 0.000, C 0.000 }
gfCNCPoint1[14022] = {X 420.3787, Y 54.1003, Z -1.3333, A 0.000, B 0.000, C 0.000 }
gfCNCPoint1[14023] = {X 421.2241, Y 54.3961, Z -1.3333, A 0.000, B 0.000, C 0.000 }
gfCNCPoint1[14024] = {X 421.9826, Y 54.8727, Z -1.3333, A 0.000, B 0.000, C 0.000 }
gfCNCPoint1[14025] = {X 422.6159, Y 55.5060, Z -1.3333, A 0.000, B 0.000, C 0.000 }
gfCNCPoint1[14026] = {X 423.0925, Y 56.2645, Z -1.3333, A 0.000, B 0.000, C 0.000 }
gfCNCPoint1[14027] = {X 423.3883, Y 57.1099, Z -1.3333, A 0.000, B 0.000, C 0.000 }
gfCNCPoint1[14028] = {X 423.4886, Y 58.0000, Z -1.3333, A 0.000, B 0.000, C 0.000 }
gfCNCPoint1[14029] = {X 423.4886, Y 58.4516, Z -1.3333, A 0.000, B 0.000, C 0.000 }
gfCNCPoint1[14030] = {X 429.4945, Y 60.7925, Z -1.3333, A 0.000, B 0.000, C 0.000 }
gfCNCPoint1[14031] = {X 458.1793, Y 72.1729, Z -1.3333, A 0.000, B 0.000, C 0.000 }
gfCNCPoint1[14032] = {X 458.1814, Y 71.5847, Z -1.3333, A 0.000, B 0.000, C 0.000 }
gfCNCPoint1[14033] = {X 458.1800, Y 63.0378, Z -1.3333, A 0.000, B 0.000, C 0.000 }
gfCNCPoint1[14034] = {X 458.1841, Y 62.9246, Z -1.3333, A 0.000, B 0.000, C 0.000 }
gfCNCPoint1[14035] = {X 458.0126, Y 62.9090, Z -1.3333, A 0.000, B 0.000, C 0.000 }
gfCNCPoint1[14036] = {X 457.8419, Y 62.8861, Z -1.3333, A 0.000, B 0.000, C 0.000 }
gfCNCPoint1[14037] = {X 456.9351, Y 62.6322, Z -1.3333, A 0.000, B 0.000, C 0.000 }
gfCNCPoint1[14038] = {X 456.1128, Y 62.1733, Z -1.3333, A 0.000, B 0.000, C 0.000 }
gfCNCPoint1[14039] = {X 455.4206, Y 61.5349, Z -1.3333, A 0.000, B 0.000, C 0.000 }
gfCNCPoint1[14040] = {X 454.8968, Y 60.7524, Z -1.3333, A 0.000, B 0.000, C 0.000 }
gfCNCPoint1[14041] = {X 454.5704, Y 59.8691, Z -1.3333, A 0.000, B 0.000, C 0.000 }
gfCNCPoint1[14042] = {X 454.4596, Y 58.9340, Z -1.3333, A 0.000, B 0.000, C 0.000 }
gfCNCPoint1[14043] = {X 454.4596, Y 58.0000, Z -1.3333, A 0.000, B 0.000, C 0.000 }
gfCNCPoint1[14044] = {X 454.5599, Y 57.1099, Z -1.3333, A 0.000, B 0.000, C 0.000 }
gfCNCPoint1[14045] = {X 454.8557, Y 56.2645, Z -1.3333, A 0.000, B 0.000, C 0.000 }
gfCNCPoint1[14046] = {X 455.3323, Y 55.5060, Z -1.3333, A 0.000, B 0.000, C 0.000 }
gfCNCPoint1[14047] = {X 455.9656, Y 54.8727, Z -1.3333, A 0.000, B 0.000, C 0.000 }
gfCNCPoint1[14048] = {X 456.7241, Y 54.3961, Z -1.3333, A 0.000, B 0.000, C 0.000 }
gfCNCPoint1[14049] = {X 457.5695, Y 54.1003, Z -1.3333, A 0.000, B 0.000, C 0.000 }
gfCNCPoint1[14050] = {X 458.4596, Y 54.0000, Z -1.3333, A 0.000, B 0.000, C 0.000 }
gfCNCPoint1[14051] = {X 475.0000, Y 54.0000, Z -1.3333, A 0.000, B 0.000, C 0.000 }
gfCNCPoint1[14052] = {X 475.8901, Y 54.1003, Z -1.3333, A 0.000, B 0.000, C 0.000 }
gfCNCPoint1[14053] = {X 476.7355, Y 54.3961, Z -1.3333, A 0.000, B 0.000, C 0.000 }
gfCNCPoint1[14054] = {X 477.4940, Y 54.8727, Z -1.3333, A 0.000, B 0.000, C 0.000 }
gfCNCPoint1[14055] = {X 478.1273, Y 55.5060, Z -1.3333, A 0.000, B 0.000, C 0.000 }
gfCNCPoint1[14056] = {X 478.6039, Y 56.2645, Z -1.3333, A 0.000, B 0.000, C 0.000 }
gfCNCPoint1[14057] = {X 478.8997, Y 57.1099, Z -1.3333, A 0.000, B 0.000, C 0.000 }
gfCNCPoint1[14058] = {X 479.0000, Y 58.0000, Z -1.3333, A 0.000, B 0.000, C 0.000 }
gfCNCPoint1[14059] = {X 478.9999, Y 58.9671, Z -1.3333, A 0.000, B 0.000, C 0.000 }
gfCNCPoint1[14060] = {X 478.9023, Y 59.8128, Z -1.3333, A 0.000, B 0.000, C 0.000 }
gfCNCPoint1[14061] = {X 478.6279, Y 60.6188, Z -1.3333, A 0.000, B 0.000, C 0.000 }
gfCNCPoint1[14062] = {X 478.1892, Y 61.3484, Z -1.3333, A 0.000, B 0.000, C 0.000 }
gfCNCPoint1[14063] = {X 477.6061, Y 61.9686, Z -1.3333, A 0.000, B 0.000, C 0.000 }
gfCNCPoint1[14064] = {X 476.9048, Y 62.4514, Z -1.3333, A 0.000, B 0.000, C 0.000 }
gfCNCPoint1[14065] = {X 476.1173, Y 62.7748, Z -1.3333, A 0.000, B 0.000, C 0.000 }
gfCNCPoint1[14066] = {X 475.2792, Y 62.9243, Z -1.3333, A 0.000, B 0.000, C 0.000 }
gfCNCPoint1[14067] = {X 475.2796, Y 93.0300, Z -1.3333, A 0.000, B 0.000, C 0.000 }
gfCNCPoint1[14068] = {X 475.7865, Y 93.1433, Z -1.3333, A 0.000, B 0.000, C 0.000 }
gfCNCPoint1[14069] = {X 476.2845, Y 93.2909, Z -1.3333, A 0.000, B 0.000, C 0.000 }
gfCNCPoint1[14070] = {X 477.0361, Y 93.6323, Z -1.3333, A 0.000, B 0.000, C 0.000 }
gfCNCPoint1[14071] = {X 477.7010, Y 94.1216, Z -1.3333, A 0.000, B 0.000, C 0.000 }
gfCNCPoint1[14072] = {X 478.2504, Y 94.7376, Z -1.3333, A 0.000, B 0.000, C 0.000 }
gfCNCPoint1[14073] = {X 478.6608, Y 95.4539, Z -1.3333, A 0.000, B 0.000, C 0.000 }
gfCNCPoint1[14074] = {X 478.9143, Y 96.2395, Z -1.3333, A 0.000, B 0.000, C 0.000 }
gfCNCPoint1[14075] = {X 479.0000, Y 97.0605, Z -1.3333, A 0.000, B 0.000, C 0.000 }
gfCNCPoint1[14076] = {X 479.0000, Y 98.0000, Z -1.3333, A 0.000, B 0.000, C 0.000 }
gfCNCPoint1[14077] = {X 478.8997, Y 98.8901, Z -1.3333, A 0.000, B 0.000, C 0.000 }
gfCNCPoint1[14078] = {X 478.6039, Y 99.7355, Z -1.3333, A 0.000, B 0.000, C 0.000 }
gfCNCPoint1[14079] = {X 478.1273, Y 100.4940, Z -1.3333, A 0.000, B 0.000, C 0.000 }
gfCNCPoint1[14080] = {X 477.4940, Y 101.1273, Z -1.3333, A 0.000, B 0.000, C 0.000 }
gfCNCPoint1[14081] = {X 476.7355, Y 101.6039, Z -1.3333, A 0.000, B 0.000, C 0.000 }
gfCNCPoint1[14082] = {X 475.8901, Y 101.8997, Z -1.3333, A 0.000, B 0.000, C 0.000 }
gfCNCPoint1[14083] = {X 475.0000, Y 102.0000, Z -1.3333, A 0.000, B 0.000, C 0.000 }
gfCNCPoint1[14084] = {X 458.4596, Y 102.0000, Z -1.3333, A 0.000, B 0.000, C 0.000 }
gfCNCPoint1[14085] = {X 457.5695, Y 101.8997, Z -1.3333, A 0.000, B 0.000, C 0.000 }
gfCNCPoint1[14086] = {X 456.7241, Y 101.6039, Z -1.3333, A 0.000, B 0.000, C 0.000 }
gfCNCPoint1[14087] = {X 455.9656, Y 101.1273, Z -1.3333, A 0.000, B 0.000, C 0.000 }
gfCNCPoint1[14088] = {X 455.3323, Y 100.4940, Z -1.3333, A 0.000, B 0.000, C 0.000 }
gfCNCPoint1[14089] = {X 454.8557, Y 99.7355, Z -1.3333, A 0.000, B 0.000, C 0.000 }
gfCNCPoint1[14090] = {X 454.5599, Y 98.8901, Z -1.3333, A 0.000, B 0.000, C 0.000 }
gfCNCPoint1[14091] = {X 454.4596, Y 98.0000, Z -1.3333, A 0.000, B 0.000, C 0.000 }
gfCNCPoint1[14092] = {X 454.4596, Y 97.0659, Z -1.3333, A 0.000, B 0.000, C 0.000 }
gfCNCPoint1[14093] = {X 454.5511, Y 96.2154, Z -1.3333, A 0.000, B 0.000, C 0.000 }
gfCNCPoint1[14094] = {X 454.8213, Y 95.4037, Z -1.3333, A 0.000, B 0.000, C 0.000 }
gfCNCPoint1[14095] = {X 455.2580, Y 94.6681, Z -1.3333, A 0.000, B 0.000, C 0.000 }
gfCNCPoint1[14096] = {X 455.8411, Y 94.0422, Z -1.3333, A 0.000, B 0.000, C 0.000 }
gfCNCPoint1[14097] = {X 456.5439, Y 93.5545, Z -1.3333, A 0.000, B 0.000, C 0.000 }
gfCNCPoint1[14098] = {X 457.3344, Y 93.2275, Z -1.3333, A 0.000, B 0.000, C 0.000 }
gfCNCPoint1[14099] = {X 458.1763, Y 93.0760, Z -1.3333, A 0.000, B 0.000, C 0.000 }
gfCNCPoint1[14100] = {X 458.1763, Y 85.3767, Z -1.3333, A 0.000, B 0.000, C 0.000 }
gfCNCPoint1[14101] = {X 444.8217, Y 80.1417, Z -1.3333, A 0.000, B 0.000, C 0.000 }
gfCNCPoint1[14102] = {X 419.7009, Y 96.4150, Z -1.3333, A 0.000, B 0.000, C 0.000 }
gfCNCPoint1[14103] = {X 419.7067, Y 97.0659, Z -1.3333, A 0.000, B 0.000, C 0.000 }
gfCNCPoint1[14104] = {X 419.7067, Y 98.0000, Z -1.3333, A 0.000, B 0.000, C 0.000 }
gfCNCPoint1[14105] = {X 419.6064, Y 98.8901, Z -1.3333, A 0.000, B 0.000, C 0.000 }
gfCNCPoint1[14106] = {X 419.3106, Y 99.7355, Z -1.3333, A 0.000, B 0.000, C 0.000 }
gfCNCPoint1[14107] = {X 418.8340, Y 100.4940, Z -1.3333, A 0.000, B 0.000, C 0.000 }
gfCNCPoint1[14108] = {X 418.2007, Y 101.1273, Z -1.3333, A 0.000, B 0.000, C 0.000 }
gfCNCPoint1[14109] = {X 417.4422, Y 101.6039, Z -1.3333, A 0.000, B 0.000, C 0.000 }
gfCNCPoint1[14110] = {X 416.5968, Y 101.8997, Z -1.3333, A 0.000, B 0.000, C 0.000 }
gfCNCPoint1[14111] = {X 415.7067, Y 102.0000, Z -1.3333, A 0.000, B 0.000, C 0.000 }
gfCNCPoint1[14112] = {X 396.4059, Y 102.0000, Z -1.3333, A 0.000, B 0.000, C 0.000 }
gfCNCPoint1[14113] = {X 395.5159, Y 101.8997, Z -1.3333, A 0.000, B 0.000, C 0.000 }
gfCNCPoint1[14114] = {X 394.6704, Y 101.6039, Z -1.3333, A 0.000, B 0.000, C 0.000 }
gfCNCPoint1[14115] = {X 393.9120, Y 101.1273, Z -1.3333, A 0.000, B 0.000, C 0.000 }
gfCNCPoint1[14116] = {X 393.2786, Y 100.4940, Z -1.3333, A 0.000, B 0.000, C 0.000 }
gfCNCPoint1[14117] = {X 392.8021, Y 99.7355, Z -1.3333, A 0.000, B 0.000, C 0.000 }
gfCNCPoint1[14118] = {X 392.5062, Y 98.8901, Z -1.3333, A 0.000, B 0.000, C 0.000 }
gfCNCPoint1[14119] = {X 392.4059, Y 98.0000, Z -1.3333, A 0.000, B 0.000, C 0.000 }
gfCNCPoint1[14120] = {X 392.4059, Y 97.0659, Z -1.3333, A 0.000, B 0.000, C 0.000 }
gfCNCPoint1[14121] = {X 392.5058, Y 96.1776, Z -1.3333, A 0.000, B 0.000, C 0.000 }
gfCNCPoint1[14122] = {X 392.8005, Y 95.3337, Z -1.3333, A 0.000, B 0.000, C 0.000 }
gfCNCPoint1[14123] = {X 393.2753, Y 94.5762, Z -1.3333, A 0.000, B 0.000, C 0.000 }
gfCNCPoint1[14124] = {X 393.9064, Y 93.9431, Z -1.3333, A 0.000, B 0.000, C 0.000 }
gfCNCPoint1[14125] = {X 394.6623, Y 93.4660, Z -1.3333, A 0.000, B 0.000, C 0.000 }
gfCNCPoint1[14126] = {X 395.5053, Y 93.1686, Z -1.3333, A 0.000, B 0.000, C 0.000 }
gfCNCPoint1[14127] = {X 396.3933, Y 93.0660, Z -1.3333, A 0.000, B 0.000, C 0.000 }
gfCNCPoint1[14128] = {X 397.3648, Y 93.0251, Z -1.3333, A 0.000, B 0.000, C 0.000 }
gfCNCPoint1[14129] = {X 398.3327, Y 92.9332, Z -1.3333, A 0.000, B 0.000, C 0.000 }
gfCNCPoint1[14130] = {X 399.0538, Y 92.7587, Z -1.3333, A 0.000, B 0.000, C 0.000 }
gfCNCPoint1[14131] = {X 399.7177, Y 92.4275, Z -1.3333, A 0.000, B 0.000, C 0.000 }
gfCNCPoint1[14132] = {X 405.3935, Y 88.7698, Z -1.3333, A 0.000, B 0.000, C 0.000 }
gfCNCPoint1[14133] = {X 413.9657, Y 83.2885, Z -1.3333, A 0.000, B 0.000, C 0.000 }
gfCNCPoint1[14134] = {X 411.7678, Y 79.8511, Z -1.3333, A 0.000, B 0.000, C 0.000 }
gfCNCPoint1[14135] = {X 411.7678, Y 79.8511, Z 1.6667, A 0.000, B 0.000, C 0.000 }
gfCNCPoint1[14136] = {X 411.7678, Y 79.8511, Z 11.0000, A 0.000, B 0.000, C 0.000 }
gfCNCPoint1[14137] = {X 466.3096, Y 28.5935, Z 11.0000, A 0.000, B 0.000, C 0.000 }
gfCNCPoint1[14138] = {X 466.3096, Y 28.5935, Z 1.6667, A 0.000, B 0.000, C 0.000 }
gfCNCPoint1[14139] = {X 466.3096, Y 28.5935, Z -1.3333, A 0.000, B 0.000, C 0.000 }
gfCNCPoint1[14140] = {X 462.2296, Y 28.5936, Z -1.3333, A 0.000, B 0.000, C 0.000 }
gfCNCPoint1[14141] = {X 462.2298, Y 40.9126, Z -1.3333, A 0.000, B 0.000, C 0.000 }
gfCNCPoint1[14142] = {X 462.2387, Y 40.9197, Z -1.3333, A 0.000, B 0.000, C 0.000 }
gfCNCPoint1[14143] = {X 462.8739, Y 41.5902, Z -1.3333, A 0.000, B 0.000, C 0.000 }
gfCNCPoint1[14144] = {X 463.3520, Y 42.3805, Z -1.3333, A 0.000, B 0.000, C 0.000 }
gfCNCPoint1[14145] = {X 463.6512, Y 43.2543, Z -1.3333, A 0.000, B 0.000, C 0.000 }
gfCNCPoint1[14146] = {X 463.7578, Y 44.1718, Z -1.3333, A 0.000, B 0.000, C 0.000 }
gfCNCPoint1[14147] = {X 463.7579, Y 45.0000, Z -1.3333, A 0.000, B 0.000, C 0.000 }
gfCNCPoint1[14148] = {X 463.6496, Y 45.9613, Z -1.3333, A 0.000, B 0.000, C 0.000 }
gfCNCPoint1[14149] = {X 463.3301, Y 46.8744, Z -1.3333, A 0.000, B 0.000, C 0.000 }
gfCNCPoint1[14150] = {X 462.8155, Y 47.6935, Z -1.3333, A 0.000, B 0.000, C 0.000 }
gfCNCPoint1[14151] = {X 462.1314, Y 48.3775, Z -1.3333, A 0.000, B 0.000, C 0.000 }
gfCNCPoint1[14152] = {X 461.3123, Y 48.8922, Z -1.3333, A 0.000, B 0.000, C 0.000 }
gfCNCPoint1[14153] = {X 460.3992, Y 49.2117, Z -1.3333, A 0.000, B 0.000, C 0.000 }
gfCNCPoint1[14154] = {X 459.4379, Y 49.3200, Z -1.3333, A 0.000, B 0.000, C 0.000 }
gfCNCPoint1[14155] = {X 452.9945, Y 49.3200, Z -1.3333, A 0.000, B 0.000, C 0.000 }
gfCNCPoint1[14156] = {X 452.0380, Y 49.2128, Z -1.3333, A 0.000, B 0.000, C 0.000 }
gfCNCPoint1[14157] = {X 451.1291, Y 48.8965, Z -1.3333, A 0.000, B 0.000, C 0.000 }
gfCNCPoint1[14158] = {X 450.3127, Y 48.3868, Z -1.3333, A 0.000, B 0.000, C 0.000 }
gfCNCPoint1[14159] = {X 449.6294, Y 47.7091, Z -1.3333, A 0.000, B 0.000, C 0.000 }
gfCNCPoint1[14160] = {X 449.1132, Y 46.8968, Z -1.3333, A 0.000, B 0.000, C 0.000 }
gfCNCPoint1[14161] = {X 448.7895, Y 45.9905, Z -1.3333, A 0.000, B 0.000, C 0.000 }
gfCNCPoint1[14162] = {X 448.6746, Y 45.0349, Z -1.3333, A 0.000, B 0.000, C 0.000 }
gfCNCPoint1[14163] = {X 448.6749, Y 44.1494, Z -1.3333, A 0.000, B 0.000, C 0.000 }
gfCNCPoint1[14164] = {X 448.7853, Y 43.2364, Z -1.3333, A 0.000, B 0.000, C 0.000 }
gfCNCPoint1[14165] = {X 449.0865, Y 42.3675, Z -1.3333, A 0.000, B 0.000, C 0.000 }
gfCNCPoint1[14166] = {X 449.5648, Y 41.5821, Z -1.3333, A 0.000, B 0.000, C 0.000 }
gfCNCPoint1[14167] = {X 450.1984, Y 40.9157, Z -1.3333, A 0.000, B 0.000, C 0.000 }
gfCNCPoint1[14168] = {X 450.1984, Y 34.4738, Z -1.3333, A 0.000, B 0.000, C 0.000 }
gfCNCPoint1[14169] = {X 447.4734, Y 34.4738, Z -1.3333, A 0.000, B 0.000, C 0.000 }
gfCNCPoint1[14170] = {X 443.1890, Y 42.8152, Z -1.3333, A 0.000, B 0.000, C 0.000 }
gfCNCPoint1[14171] = {X 443.1942, Y 42.8290, Z -1.3333, A 0.000, B 0.000, C 0.000 }
gfCNCPoint1[14172] = {X 443.3604, Y 43.4907, Z -1.3333, A 0.000, B 0.000, C 0.000 }
gfCNCPoint1[14173] = {X 443.4203, Y 44.1703, Z -1.3333, A 0.000, B 0.000, C 0.000 }
gfCNCPoint1[14174] = {X 443.4205, Y 45.0000, Z -1.3333, A 0.000, B 0.000, C 0.000 }
gfCNCPoint1[14175] = {X 443.3122, Y 45.9613, Z -1.3333, A 0.000, B 0.000, C 0.000 }
gfCNCPoint1[14176] = {X 442.9927, Y 46.8744, Z -1.3333, A 0.000, B 0.000, C 0.000 }
gfCNCPoint1[14177] = {X 442.4780, Y 47.6935, Z -1.3333, A 0.000, B 0.000, C 0.000 }
gfCNCPoint1[14178] = {X 441.7939, Y 48.3775, Z -1.3333, A 0.000, B 0.000, C 0.000 }
gfCNCPoint1[14179] = {X 440.9748, Y 48.8922, Z -1.3333, A 0.000, B 0.000, C 0.000 }
gfCNCPoint1[14180] = {X 440.0618, Y 49.2117, Z -1.3333, A 0.000, B 0.000, C 0.000 }
gfCNCPoint1[14181] = {X 439.1005, Y 49.3200, Z -1.3333, A 0.000, B 0.000, C 0.000 }
gfCNCPoint1[14182] = {X 432.5144, Y 49.3200, Z -1.3333, A 0.000, B 0.000, C 0.000 }
gfCNCPoint1[14183] = {X 431.5531, Y 49.2117, Z -1.3333, A 0.000, B 0.000, C 0.000 }
gfCNCPoint1[14184] = {X 430.6401, Y 48.8922, Z -1.3333, A 0.000, B 0.000, C 0.000 }
gfCNCPoint1[14185] = {X 429.8210, Y 48.3775, Z -1.3333, A 0.000, B 0.000, C 0.000 }
gfCNCPoint1[14186] = {X 429.1369, Y 47.6935, Z -1.3333, A 0.000, B 0.000, C 0.000 }
gfCNCPoint1[14187] = {X 428.6223, Y 46.8745, Z -1.3333, A 0.000, B 0.000, C 0.000 }
gfCNCPoint1[14188] = {X 428.3027, Y 45.9614, Z -1.3333, A 0.000, B 0.000, C 0.000 }
gfCNCPoint1[14189] = {X 428.1944, Y 45.0001, Z -1.3333, A 0.000, B 0.000, C 0.000 }
gfCNCPoint1[14190] = {X 428.1948, Y 44.1494, Z -1.3333, A 0.000, B 0.000, C 0.000 }
gfCNCPoint1[14191] = {X 428.2925, Y 43.2935, Z -1.3333, A 0.000, B 0.000, C 0.000 }
gfCNCPoint1[14192] = {X 428.5580, Y 42.4740, Z -1.3333, A 0.000, B 0.000, C 0.000 }
gfCNCPoint1[14193] = {X 428.9809, Y 41.7236, Z -1.3333, A 0.000, B 0.000, C 0.000 }
gfCNCPoint1[14194] = {X 429.5442, Y 41.0719, Z -1.3333, A 0.000, B 0.000, C 0.000 }
gfCNCPoint1[14195] = {X 430.2256, Y 40.5449, Z -1.3333, A 0.000, B 0.000, C 0.000 }
gfCNCPoint1[14196] = {X 430.9981, Y 40.1637, Z -1.3333, A 0.000, B 0.000, C 0.000 }
gfCNCPoint1[14197] = {X 434.9875, Y 32.3548, Z -1.3333, A 0.000, B 0.000, C 0.000 }
gfCNCPoint1[14198] = {X 433.8177, Y 31.5683, Z -1.3333, A 0.000, B 0.000, C 0.000 }
gfCNCPoint1[14199] = {X 432.7548, Y 30.6426, Z -1.3333, A 0.000, B 0.000, C 0.000 }
gfCNCPoint1[14200] = {X 431.8151, Y 29.5919, Z -1.3333, A 0.000, B 0.000, C 0.000 }
gfCNCPoint1[14201] = {X 431.0133, Y 28.4327, Z -1.3333, A 0.000, B 0.000, C 0.000 }
gfCNCPoint1[14202] = {X 430.3617, Y 27.1827, Z -1.3333, A 0.000, B 0.000, C 0.000 }
gfCNCPoint1[14203] = {X 429.8706, Y 25.8615, Z -1.3333, A 0.000, B 0.000, C 0.000 }
gfCNCPoint1[14204] = {X 429.4515, Y 24.0500, Z -1.3333, A 0.000, B 0.000, C 0.000 }
gfCNCPoint1[14205] = {X 429.2379, Y 22.2029, Z -1.3333, A 0.000, B 0.000, C 0.000 }
gfCNCPoint1[14206] = {X 429.2325, Y 20.3436, Z -1.3333, A 0.000, B 0.000, C 0.000 }
gfCNCPoint1[14207] = {X 429.4354, Y 18.4953, Z -1.3333, A 0.000, B 0.000, C 0.000 }
gfCNCPoint1[14208] = {X 429.8440, Y 16.6814, Z -1.3333, A 0.000, B 0.000, C 0.000 }
gfCNCPoint1[14209] = {X 430.3654, Y 15.2117, Z -1.3333, A 0.000, B 0.000, C 0.000 }
gfCNCPoint1[14210] = {X 431.0761, Y 13.8236, Z -1.3333, A 0.000, B 0.000, C 0.000 }
gfCNCPoint1[14211] = {X 431.9638, Y 12.5415, Z -1.3333, A 0.000, B 0.000, C 0.000 }
gfCNCPoint1[14212] = {X 433.0130, Y 11.3877, Z -1.3333, A 0.000, B 0.000, C 0.000 }
gfCNCPoint1[14213] = {X 434.2052, Y 10.3825, Z -1.3333, A 0.000, B 0.000, C 0.000 }
gfCNCPoint1[14214] = {X 435.5197, Y 9.5433, Z -1.3333, A 0.000, B 0.000, C 0.000 }
gfCNCPoint1[14215] = {X 436.9334, Y 8.8850, Z -1.3333, A 0.000, B 0.000, C 0.000 }
gfCNCPoint1[14216] = {X 438.4216, Y 8.4190, Z -1.3333, A 0.000, B 0.000, C 0.000 }
gfCNCPoint1[14217] = {X 440.0467, Y 8.1098, Z -1.3333, A 0.000, B 0.000, C 0.000 }
gfCNCPoint1[14218] = {X 441.6910, Y 7.9284, Z -1.3333, A 0.000, B 0.000, C 0.000 }
gfCNCPoint1[14219] = {X 443.3444, Y 7.8759, Z -1.3333, A 0.000, B 0.000, C 0.000 }
gfCNCPoint1[14220] = {X 444.0357, Y 7.8719, Z -1.3333, A 0.000, B 0.000, C 0.000 }
gfCNCPoint1[14221] = {X 459.4465, Y 7.8719, Z -1.3333, A 0.000, B 0.000, C 0.000 }
gfCNCPoint1[14222] = {X 460.4059, Y 7.9800, Z -1.3333, A 0.000, B 0.000, C 0.000 }
gfCNCPoint1[14223] = {X 461.3172, Y 8.2989, Z -1.3333, A 0.000, B 0.000, C 0.000 }
gfCNCPoint1[14224] = {X 462.1346, Y 8.8125, Z -1.3333, A 0.000, B 0.000, C 0.000 }
gfCNCPoint1[14225] = {X 462.8173, Y 9.4952, Z -1.3333, A 0.000, B 0.000, C 0.000 }
gfCNCPoint1[14226] = {X 463.3310, Y 10.3127, Z -1.3333, A 0.000, B 0.000, C 0.000 }
gfCNCPoint1[14227] = {X 463.6498, Y 11.2240, Z -1.3333, A 0.000, B 0.000, C 0.000 }
gfCNCPoint1[14228] = {X 463.7579, Y 12.1834, Z -1.3333, A 0.000, B 0.000, C 0.000 }
gfCNCPoint1[14229] = {X 463.7579, Y 12.9781, Z -1.3333, A 0.000, B 0.000, C 0.000 }
gfCNCPoint1[14230] = {X 463.6565, Y 13.9083, Z -1.3333, A 0.000, B 0.000, C 0.000 }
gfCNCPoint1[14231] = {X 463.3571, Y 14.7949, Z -1.3333, A 0.000, B 0.000, C 0.000 }
gfCNCPoint1[14232] = {X 462.8739, Y 15.5961, Z -1.3333, A 0.000, B 0.000, C 0.000 }
gfCNCPoint1[14233] = {X 462.2294, Y 16.2746, Z -1.3333, A 0.000, B 0.000, C 0.000 }
gfCNCPoint1[14234] = {X 462.2296, Y 28.5936, Z -1.3333, A 0.000, B 0.000, C 0.000 }
gfCNCPoint1[14235] = {X 466.2296, Y 28.5935, Z -1.3333, A 0.000, B 0.000, C 0.000 }
gfCNCPoint1[14236] = {X 462.1496, Y 28.5936, Z -1.3333, A 0.000, B 0.000, C 0.000 }
gfCNCPoint1[14237] = {X 462.1498, Y 40.9509, Z -1.3333, A 0.000, B 0.000, C 0.000 }
gfCNCPoint1[14238] = {X 462.1877, Y 40.9813, Z -1.3333, A 0.000, B 0.000, C 0.000 }
gfCNCPoint1[14239] = {X 462.8107, Y 41.6394, Z -1.3333, A 0.000, B 0.000, C 0.000 }
gfCNCPoint1[14240] = {X 463.2797, Y 42.4148, Z -1.3333, A 0.000, B 0.000, C 0.000 }
gfCNCPoint1[14241] = {X 463.5732, Y 43.2723, Z -1.3333, A 0.000, B 0.000, C 0.000 }
gfCNCPoint1[14242] = {X 463.6778, Y 44.1724, Z -1.3333, A 0.000, B 0.000, C 0.000 }
gfCNCPoint1[14243] = {X 463.6779, Y 45.0000, Z -1.3333, A 0.000, B 0.000, C 0.000 }
gfCNCPoint1[14244] = {X 463.5716, Y 45.9435, Z -1.3333, A 0.000, B 0.000, C 0.000 }
gfCNCPoint1[14245] = {X 463.2580, Y 46.8397, Z -1.3333, A 0.000, B 0.000, C 0.000 }
gfCNCPoint1[14246] = {X 462.7529, Y 47.6436, Z -1.3333, A 0.000, B 0.000, C 0.000 }
gfCNCPoint1[14247] = {X 462.0815, Y 48.3150, Z -1.3333, A 0.000, B 0.000, C 0.000 }
gfCNCPoint1[14248] = {X 461.2776, Y 48.8201, Z -1.3333, A 0.000, B 0.000, C 0.000 }
gfCNCPoint1[14249] = {X 460.3814, Y 49.1337, Z -1.3333, A 0.000, B 0.000, C 0.000 }
gfCNCPoint1[14250] = {X 459.4379, Y 49.2400, Z -1.3333, A 0.000, B 0.000, C 0.000 }
gfCNCPoint1[14251] = {X 452.9945, Y 49.2400, Z -1.3333, A 0.000, B 0.000, C 0.000 }
gfCNCPoint1[14252] = {X 452.0558, Y 49.1348, Z -1.3333, A 0.000, B 0.000, C 0.000 }
gfCNCPoint1[14253] = {X 451.1636, Y 48.8243, Z -1.3333, A 0.000, B 0.000, C 0.000 }
gfCNCPoint1[14254] = {X 450.3624, Y 48.3241, Z -1.3333, A 0.000, B 0.000, C 0.000 }
gfCNCPoint1[14255] = {X 449.6918, Y 47.6589, Z -1.3333, A 0.000, B 0.000, C 0.000 }
gfCNCPoint1[14256] = {X 449.1851, Y 46.8617, Z -1.3333, A 0.000, B 0.000, C 0.000 }
gfCNCPoint1[14257] = {X 448.8674, Y 45.9721, Z -1.3333, A 0.000, B 0.000, C 0.000 }
gfCNCPoint1[14258] = {X 448.7546, Y 45.0343, Z -1.3333, A 0.000, B 0.000, C 0.000 }
gfCNCPoint1[14259] = {X 448.7549, Y 44.1505, Z -1.3333, A 0.000, B 0.000, C 0.000 }
gfCNCPoint1[14260] = {X 448.8654, Y 43.2454, Z -1.3333, A 0.000, B 0.000, C 0.000 }
gfCNCPoint1[14261] = {X 449.1668, Y 42.3850, Z -1.3333, A 0.000, B 0.000, C 0.000 }
gfCNCPoint1[14262] = {X 449.6452, Y 41.6088, Z -1.3333, A 0.000, B 0.000, C 0.000 }
gfCNCPoint1[14263] = {X 450.2784, Y 40.9529, Z -1.3333, A 0.000, B 0.000, C 0.000 }
gfCNCPoint1[14264] = {X 450.2784, Y 34.3938, Z -1.3333, A 0.000, B 0.000, C 0.000 }
gfCNCPoint1[14265] = {X 447.4245, Y 34.3938, Z -1.3333, A 0.000, B 0.000, C 0.000 }
gfCNCPoint1[14266] = {X 443.1017, Y 42.8102, Z -1.3333, A 0.000, B 0.000, C 0.000 }
gfCNCPoint1[14267] = {X 443.1188, Y 42.8559, Z -1.3333, A 0.000, B 0.000, C 0.000 }
gfCNCPoint1[14268] = {X 443.2816, Y 43.5047, Z -1.3333, A 0.000, B 0.000, C 0.000 }
gfCNCPoint1[14269] = {X 443.3403, Y 44.1710, Z -1.3333, A 0.000, B 0.000, C 0.000 }
gfCNCPoint1[14270] = {X 443.3405, Y 45.0000, Z -1.3333, A 0.000, B 0.000, C 0.000 }
gfCNCPoint1[14271] = {X 443.2342, Y 45.9435, Z -1.3333, A 0.000, B 0.000, C 0.000 }
gfCNCPoint1[14272] = {X 442.9206, Y 46.8397, Z -1.3333, A 0.000, B 0.000, C 0.000 }
gfCNCPoint1[14273] = {X 442.4154, Y 47.6436, Z -1.3333, A 0.000, B 0.000, C 0.000 }
gfCNCPoint1[14274] = {X 441.7441, Y 48.3150, Z -1.3333, A 0.000, B 0.000, C 0.000 }
gfCNCPoint1[14275] = {X 440.9401, Y 48.8201, Z -1.3333, A 0.000, B 0.000, C 0.000 }
gfCNCPoint1[14276] = {X 440.0440, Y 49.1337, Z -1.3333, A 0.000, B 0.000, C 0.000 }
gfCNCPoint1[14277] = {X 439.1005, Y 49.2400, Z -1.3333, A 0.000, B 0.000, C 0.000 }
gfCNCPoint1[14278] = {X 432.5144, Y 49.2400, Z -1.3333, A 0.000, B 0.000, C 0.000 }
gfCNCPoint1[14279] = {X 431.5709, Y 49.1337, Z -1.3333, A 0.000, B 0.000, C 0.000 }
gfCNCPoint1[14280] = {X 430.6748, Y 48.8201, Z -1.3333, A 0.000, B 0.000, C 0.000 }
gfCNCPoint1[14281] = {X 429.8708, Y 48.3150, Z -1.3333, A 0.000, B 0.000, C 0.000 }
gfCNCPoint1[14282] = {X 429.1995, Y 47.6436, Z -1.3333, A 0.000, B 0.000, C 0.000 }
gfCNCPoint1[14283] = {X 428.6943, Y 46.8397, Z -1.3333, A 0.000, B 0.000, C 0.000 }
gfCNCPoint1[14284] = {X 428.3807, Y 45.9436, Z -1.3333, A 0.000, B 0.000, C 0.000 }
gfCNCPoint1[14285] = {X 428.2744, Y 45.0001, Z -1.3333, A 0.000, B 0.000, C 0.000 }
gfCNCPoint1[14286] = {X 428.2748, Y 44.1505, Z -1.3333, A 0.000, B 0.000, C 0.000 }
gfCNCPoint1[14287] = {X 428.3718, Y 43.3054, Z -1.3333, A 0.000, B 0.000, C 0.000 }
gfCNCPoint1[14288] = {X 428.6354, Y 42.4967, Z -1.3333, A 0.000, B 0.000, C 0.000 }
gfCNCPoint1[14289] = {X 429.0552, Y 41.7570, Z -1.3333, A 0.000, B 0.000, C 0.000 }
gfCNCPoint1[14290] = {X 429.6142, Y 41.1158, Z -1.3333, A 0.000, B 0.000, C 0.000 }
gfCNCPoint1[14291] = {X 430.2899, Y 40.5992, Z -1.3333, A 0.000, B 0.000, C 0.000 }
gfCNCPoint1[14292] = {X 431.0551, Y 40.2278, Z -1.3333, A 0.000, B 0.000, C 0.000 }
gfCNCPoint1[14293] = {X 435.0932, Y 32.3237, Z -1.3333, A 0.000, B 0.000, C 0.000 }
gfCNCPoint1[14294] = {X 433.9165, Y 31.5430, Z -1.3333, A 0.000, B 0.000, C 0.000 }
gfCNCPoint1[14295] = {X 432.8469, Y 30.6209, Z -1.3333, A 0.000, B 0.000, C 0.000 }
gfCNCPoint1[14296] = {X 431.9013, Y 29.5721, Z -1.3333, A 0.000, B 0.000, C 0.000 }
gfCNCPoint1[14297] = {X 431.0948, Y 28.4129, Z -1.3333, A 0.000, B 0.000, C 0.000 }
gfCNCPoint1[14298] = {X 430.4400, Y 27.1617, Z -1.3333, A 0.000, B 0.000, C 0.000 }
gfCNCPoint1[14299] = {X 429.9472, Y 25.8383, Z -1.3333, A 0.000, B 0.000, C 0.000 }
gfCNCPoint1[14300] = {X 429.5302, Y 24.0357, Z -1.3333, A 0.000, B 0.000, C 0.000 }
gfCNCPoint1[14301] = {X 429.3177, Y 22.1977, Z -1.3333, A 0.000, B 0.000, C 0.000 }
gfCNCPoint1[14302] = {X 429.3124, Y 20.3474, Z -1.3333, A 0.000, B 0.000, C 0.000 }
gfCNCPoint1[14303] = {X 429.5144, Y 18.5082, Z -1.3333, A 0.000, B 0.000, C 0.000 }
gfCNCPoint1[14304] = {X 429.9210, Y 16.7032, Z -1.3333, A 0.000, B 0.000, C 0.000 }
gfCNCPoint1[14305] = {X 430.4388, Y 15.2434, Z -1.3333, A 0.000, B 0.000, C 0.000 }
gfCNCPoint1[14306] = {X 431.1447, Y 13.8648, Z -1.3333, A 0.000, B 0.000, C 0.000 }
gfCNCPoint1[14307] = {X 432.0264, Y 12.5913, Z -1.3333, A 0.000, B 0.000, C 0.000 }
gfCNCPoint1[14308] = {X 433.0684, Y 11.4454, Z -1.3333, A 0.000, B 0.000, C 0.000 }
gfCNCPoint1[14309] = {X 434.2526, Y 10.4469, Z -1.3333, A 0.000, B 0.000, C 0.000 }
gfCNCPoint1[14310] = {X 435.5581, Y 9.6135, Z -1.3333, A 0.000, B 0.000, C 0.000 }
gfCNCPoint1[14311] = {X 436.9623, Y 8.9596, Z -1.3333, A 0.000, B 0.000, C 0.000 }
gfCNCPoint1[14312] = {X 438.4404, Y 8.4968, Z -1.3333, A 0.000, B 0.000, C 0.000 }
gfCNCPoint1[14313] = {X 440.0593, Y 8.1888, Z -1.3333, A 0.000, B 0.000, C 0.000 }
gfCNCPoint1[14314] = {X 441.6973, Y 8.0082, Z -1.3333, A 0.000, B 0.000, C 0.000 }
gfCNCPoint1[14315] = {X 443.3444, Y 7.9560, Z -1.3333, A 0.000, B 0.000, C 0.000 }
gfCNCPoint1[14316] = {X 444.0360, Y 7.9519, Z -1.3333, A 0.000, B 0.000, C 0.000 }
gfCNCPoint1[14317] = {X 459.4465, Y 7.9519, Z -1.3333, A 0.000, B 0.000, C 0.000 }
gfCNCPoint1[14318] = {X 460.3881, Y 8.0580, Z -1.3333, A 0.000, B 0.000, C 0.000 }
gfCNCPoint1[14319] = {X 461.2824, Y 8.3709, Z -1.3333, A 0.000, B 0.000, C 0.000 }
gfCNCPoint1[14320] = {X 462.0848, Y 8.8751, Z -1.3333, A 0.000, B 0.000, C 0.000 }
gfCNCPoint1[14321] = {X 462.7548, Y 9.5451, Z -1.3333, A 0.000, B 0.000, C 0.000 }
gfCNCPoint1[14322] = {X 463.2589, Y 10.3474, Z -1.3333, A 0.000, B 0.000, C 0.000 }
gfCNCPoint1[14323] = {X 463.5718, Y 11.2418, Z -1.3333, A 0.000, B 0.000, C 0.000 }
gfCNCPoint1[14324] = {X 463.6779, Y 12.1834, Z -1.3333, A 0.000, B 0.000, C 0.000 }
gfCNCPoint1[14325] = {X 463.6779, Y 12.9781, Z -1.3333, A 0.000, B 0.000, C 0.000 }
gfCNCPoint1[14326] = {X 463.5764, Y 13.9001, Z -1.3333, A 0.000, B 0.000, C 0.000 }
gfCNCPoint1[14327] = {X 463.2767, Y 14.7780, Z -1.3333, A 0.000, B 0.000, C 0.000 }
gfCNCPoint1[14328] = {X 462.7934, Y 15.5696, Z -1.3333, A 0.000, B 0.000, C 0.000 }
gfCNCPoint1[14329] = {X 462.1494, Y 16.2373, Z -1.3333, A 0.000, B 0.000, C 0.000 }
gfCNCPoint1[14330] = {X 462.1496, Y 28.5936, Z -1.3333, A 0.000, B 0.000, C 0.000 }
gfCNCPoint1[14331] = {X 466.1496, Y 28.5935, Z -1.3333, A 0.000, B 0.000, C 0.000 }
gfCNCPoint1[14332] = {X 462.0696, Y 28.5936, Z -1.3333, A 0.000, B 0.000, C 0.000 }
gfCNCPoint1[14333] = {X 462.0698, Y 40.9892, Z -1.3333, A 0.000, B 0.000, C 0.000 }
gfCNCPoint1[14334] = {X 462.1367, Y 41.0430, Z -1.3333, A 0.000, B 0.000, C 0.000 }
gfCNCPoint1[14335] = {X 462.7476, Y 41.6886, Z -1.3333, A 0.000, B 0.000, C 0.000 }
gfCNCPoint1[14336] = {X 463.2075, Y 42.4492, Z -1.3333, A 0.000, B 0.000, C 0.000 }
gfCNCPoint1[14337] = {X 463.4953, Y 43.2902, Z -1.3333, A 0.000, B 0.000, C 0.000 }
gfCNCPoint1[14338] = {X 463.5978, Y 44.1731, Z -1.3333, A 0.000, B 0.000, C 0.000 }
gfCNCPoint1[14339] = {X 463.5979, Y 45.0000, Z -1.3333, A 0.000, B 0.000, C 0.000 }
gfCNCPoint1[14340] = {X 463.4936, Y 45.9257, Z -1.3333, A 0.000, B 0.000, C 0.000 }
gfCNCPoint1[14341] = {X 463.1860, Y 46.8050, Z -1.3333, A 0.000, B 0.000, C 0.000 }
gfCNCPoint1[14342] = {X 462.6904, Y 47.5937, Z -1.3333, A 0.000, B 0.000, C 0.000 }
gfCNCPoint1[14343] = {X 462.0317, Y 48.2524, Z -1.3333, A 0.000, B 0.000, C 0.000 }
gfCNCPoint1[14344] = {X 461.2429, Y 48.7480, Z -1.3333, A 0.000, B 0.000, C 0.000 }
gfCNCPoint1[14345] = {X 460.3636, Y 49.0557, Z -1.3333, A 0.000, B 0.000, C 0.000 }
gfCNCPoint1[14346] = {X 459.4379, Y 49.1600, Z -1.3333, A 0.000, B 0.000, C 0.000 }
gfCNCPoint1[14347] = {X 452.9945, Y 49.1600, Z -1.3333, A 0.000, B 0.000, C 0.000 }
gfCNCPoint1[14348] = {X 452.0735, Y 49.0568, Z -1.3333, A 0.000, B 0.000, C 0.000 }
gfCNCPoint1[14349] = {X 451.1982, Y 48.7522, Z -1.3333, A 0.000, B 0.000, C 0.000 }
gfCNCPoint1[14350] = {X 450.4120, Y 48.2614, Z -1.3333, A 0.000, B 0.000, C 0.000 }
gfCNCPoint1[14351] = {X 449.7541, Y 47.6087, Z -1.3333, A 0.000, B 0.000, C 0.000 }
gfCNCPoint1[14352] = {X 449.2569, Y 46.8266, Z -1.3333, A 0.000, B 0.000, C 0.000 }
gfCNCPoint1[14353] = {X 448.9453, Y 45.9538, Z -1.3333, A 0.000, B 0.000, C 0.000 }
gfCNCPoint1[14354] = {X 448.8346, Y 45.0336, Z -1.3333, A 0.000, B 0.000, C 0.000 }
gfCNCPoint1[14355] = {X 448.8349, Y 44.1516, Z -1.3333, A 0.000, B 0.000, C 0.000 }
gfCNCPoint1[14356] = {X 448.9454, Y 43.2545, Z -1.3333, A 0.000, B 0.000, C 0.000 }
gfCNCPoint1[14357] = {X 449.2471, Y 42.4026, Z -1.3333, A 0.000, B 0.000, C 0.000 }
gfCNCPoint1[14358] = {X 449.7256, Y 41.6358, Z -1.3333, A 0.000, B 0.000, C 0.000 }
gfCNCPoint1[14359] = {X 450.3584, Y 40.9906, Z -1.3333, A 0.000, B 0.000, C 0.000 }
gfCNCPoint1[14360] = {X 450.3584, Y 34.3138, Z -1.3333, A 0.000, B 0.000, C 0.000 }
gfCNCPoint1[14361] = {X 447.3757, Y 34.3138, Z -1.3333, A 0.000, B 0.000, C 0.000 }
gfCNCPoint1[14362] = {X 443.0143, Y 42.8051, Z -1.3333, A 0.000, B 0.000, C 0.000 }
gfCNCPoint1[14363] = {X 443.0434, Y 42.8827, Z -1.3333, A 0.000, B 0.000, C 0.000 }
gfCNCPoint1[14364] = {X 443.2028, Y 43.5186, Z -1.3333, A 0.000, B 0.000, C 0.000 }
gfCNCPoint1[14365] = {X 443.2603, Y 44.1717, Z -1.3333, A 0.000, B 0.000, C 0.000 }
gfCNCPoint1[14366] = {X 443.2605, Y 45.0000, Z -1.3333, A 0.000, B 0.000, C 0.000 }
gfCNCPoint1[14367] = {X 443.1562, Y 45.9257, Z -1.3333, A 0.000, B 0.000, C 0.000 }
gfCNCPoint1[14368] = {X 442.8485, Y 46.8050, Z -1.3333, A 0.000, B 0.000, C 0.000 }
gfCNCPoint1[14369] = {X 442.3529, Y 47.5937, Z -1.3333, A 0.000, B 0.000, C 0.000 }
gfCNCPoint1[14370] = {X 441.6942, Y 48.2524, Z -1.3333, A 0.000, B 0.000, C 0.000 }
gfCNCPoint1[14371] = {X 440.9054, Y 48.7480, Z -1.3333, A 0.000, B 0.000, C 0.000 }
gfCNCPoint1[14372] = {X 440.0262, Y 49.0557, Z -1.3333, A 0.000, B 0.000, C 0.000 }
gfCNCPoint1[14373] = {X 439.1005, Y 49.1600, Z -1.3333, A 0.000, B 0.000, C 0.000 }
gfCNCPoint1[14374] = {X 432.5144, Y 49.1600, Z -1.3333, A 0.000, B 0.000, C 0.000 }
gfCNCPoint1[14375] = {X 431.5887, Y 49.0557, Z -1.3333, A 0.000, B 0.000, C 0.000 }
gfCNCPoint1[14376] = {X 430.7095, Y 48.7480, Z -1.3333, A 0.000, B 0.000, C 0.000 }
gfCNCPoint1[14377] = {X 429.9207, Y 48.2524, Z -1.3333, A 0.000, B 0.000, C 0.000 }
gfCNCPoint1[14378] = {X 429.2620, Y 47.5937, Z -1.3333, A 0.000, B 0.000, C 0.000 }
gfCNCPoint1[14379] = {X 428.7664, Y 46.8050, Z -1.3333, A 0.000, B 0.000, C 0.000 }
gfCNCPoint1[14380] = {X 428.4587, Y 45.9257, Z -1.3333, A 0.000, B 0.000, C 0.000 }
gfCNCPoint1[14381] = {X 428.3544, Y 45.0000, Z -1.3333, A 0.000, B 0.000, C 0.000 }
gfCNCPoint1[14382] = {X 428.3548, Y 44.1516, Z -1.3333, A 0.000, B 0.000, C 0.000 }
gfCNCPoint1[14383] = {X 428.4510, Y 43.3174, Z -1.3333, A 0.000, B 0.000, C 0.000 }
gfCNCPoint1[14384] = {X 428.7128, Y 42.5195, Z -1.3333, A 0.000, B 0.000, C 0.000 }
gfCNCPoint1[14385] = {X 429.1295, Y 41.7905, Z -1.3333, A 0.000, B 0.000, C 0.000 }
gfCNCPoint1[14386] = {X 429.6841, Y 41.1600, Z -1.3333, A 0.000, B 0.000, C 0.000 }
gfCNCPoint1[14387] = {X 430.3541, Y 40.6537, Z -1.3333, A 0.000, B 0.000, C 0.000 }
gfCNCPoint1[14388] = {X 431.1120, Y 40.2923, Z -1.3333, A 0.000, B 0.000, C 0.000 }
gfCNCPoint1[14389] = {X 435.1992, Y 32.2921, Z -1.3333, A 0.000, B 0.000, C 0.000 }
gfCNCPoint1[14390] = {X 434.0154, Y 31.5174, Z -1.3333, A 0.000, B 0.000, C 0.000 }
gfCNCPoint1[14391] = {X 432.9391, Y 30.5991, Z -1.3333, A 0.000, B 0.000, C 0.000 }
gfCNCPoint1[14392] = {X 431.9877, Y 29.5521, Z -1.3333, A 0.000, B 0.000, C 0.000 }
gfCNCPoint1[14393] = {X 431.1764, Y 28.3931, Z -1.3333, A 0.000, B 0.000, C 0.000 }
gfCNCPoint1[14394] = {X 430.5182, Y 27.1407, Z -1.3333, A 0.000, B 0.000, C 0.000 }
gfCNCPoint1[14395] = {X 430.0237, Y 25.8152, Z -1.3333, A 0.000, B 0.000, C 0.000 }
gfCNCPoint1[14396] = {X 429.6089, Y 24.0214, Z -1.3333, A 0.000, B 0.000, C 0.000 }
gfCNCPoint1[14397] = {X 429.3975, Y 22.1924, Z -1.3333, A 0.000, B 0.000, C 0.000 }
gfCNCPoint1[14398] = {X 429.3923, Y 20.3513, Z -1.3333, A 0.000, B 0.000, C 0.000 }
gfCNCPoint1[14399] = {X 429.5933, Y 18.5212, Z -1.3333, A 0.000, B 0.000, C 0.000 }
gfCNCPoint1[14400] = {X 429.9980, Y 16.7251, Z -1.3333, A 0.000, B 0.000, C 0.000 }
gfCNCPoint1[14401] = {X 430.5122, Y 15.2752, Z -1.3333, A 0.000, B 0.000, C 0.000 }
gfCNCPoint1[14402] = {X 431.2133, Y 13.9060, Z -1.3333, A 0.000, B 0.000, C 0.000 }
gfCNCPoint1[14403] = {X 432.0890, Y 12.6412, Z -1.3333, A 0.000, B 0.000, C 0.000 }
gfCNCPoint1[14404] = {X 433.1239, Y 11.5030, Z -1.3333, A 0.000, B 0.000, C 0.000 }
gfCNCPoint1[14405] = {X 434.3000, Y 10.5114, Z -1.3333, A 0.000, B 0.000, C 0.000 }
gfCNCPoint1[14406] = {X 435.5966, Y 9.6836, Z -1.3333, A 0.000, B 0.000, C 0.000 }
gfCNCPoint1[14407] = {X 436.9911, Y 9.0342, Z -1.3333, A 0.000, B 0.000, C 0.000 }
gfCNCPoint1[14408] = {X 438.4592, Y 8.5746, Z -1.3333, A 0.000, B 0.000, C 0.000 }
gfCNCPoint1[14409] = {X 440.0719, Y 8.2678, Z -1.3333, A 0.000, B 0.000, C 0.000 }
gfCNCPoint1[14410] = {X 441.7035, Y 8.0879, Z -1.3333, A 0.000, B 0.000, C 0.000 }
gfCNCPoint1[14411] = {X 443.3443, Y 8.0360, Z -1.3333, A 0.000, B 0.000, C 0.000 }
gfCNCPoint1[14412] = {X 444.0362, Y 8.0319, Z -1.3333, A 0.000, B 0.000, C 0.000 }
gfCNCPoint1[14413] = {X 459.4465, Y 8.0319, Z -1.3333, A 0.000, B 0.000, C 0.000 }
gfCNCPoint1[14414] = {X 460.3703, Y 8.1360, Z -1.3333, A 0.000, B 0.000, C 0.000 }
gfCNCPoint1[14415] = {X 461.2477, Y 8.4430, Z -1.3333, A 0.000, B 0.000, C 0.000 }
gfCNCPoint1[14416] = {X 462.0349, Y 8.9376, Z -1.3333, A 0.000, B 0.000, C 0.000 }
gfCNCPoint1[14417] = {X 462.6922, Y 9.5950, Z -1.3333, A 0.000, B 0.000, C 0.000 }
gfCNCPoint1[14418] = {X 463.1868, Y 10.3821, Z -1.3333, A 0.000, B 0.000, C 0.000 }
gfCNCPoint1[14419] = {X 463.4939, Y 11.2596, Z -1.3333, A 0.000, B 0.000, C 0.000 }
gfCNCPoint1[14420] = {X 463.5979, Y 12.1834, Z -1.3333, A 0.000, B 0.000, C 0.000 }
gfCNCPoint1[14421] = {X 463.5979, Y 12.9781, Z -1.3333, A 0.000, B 0.000, C 0.000 }
gfCNCPoint1[14422] = {X 463.5022, Y 13.8654, Z -1.3333, A 0.000, B 0.000, C 0.000 }
gfCNCPoint1[14423] = {X 463.2194, Y 14.7118, Z -1.3333, A 0.000, B 0.000, C 0.000 }
gfCNCPoint1[14424] = {X 462.7626, Y 15.4785, Z -1.3333, A 0.000, B 0.000, C 0.000 }
gfCNCPoint1[14425] = {X 462.1528, Y 16.1300, Z -1.3333, A 0.000, B 0.000, C 0.000 }
gfCNCPoint1[14426] = {X 462.0694, Y 16.2000, Z -1.3333, A 0.000, B 0.000, C 0.000 }
gfCNCPoint1[14427] = {X 462.0696, Y 28.5936, Z -1.3333, A 0.000, B 0.000, C 0.000 }
gfCNCPoint1[14428] = {X 466.0696, Y 28.5935, Z -1.3333, A 0.000, B 0.000, C 0.000 }
gfCNCPoint1[14429] = {X 461.9896, Y 28.5936, Z -1.3333, A 0.000, B 0.000, C 0.000 }
gfCNCPoint1[14430] = {X 461.9898, Y 41.0276, Z -1.3333, A 0.000, B 0.000, C 0.000 }
gfCNCPoint1[14431] = {X 462.0856, Y 41.1046, Z -1.3333, A 0.000, B 0.000, C 0.000 }
gfCNCPoint1[14432] = {X 462.6845, Y 41.7377, Z -1.3333, A 0.000, B 0.000, C 0.000 }
gfCNCPoint1[14433] = {X 463.1352, Y 42.4836, Z -1.3333, A 0.000, B 0.000, C 0.000 }
gfCNCPoint1[14434] = {X 463.4173, Y 43.3081, Z -1.3333, A 0.000, B 0.000, C 0.000 }
gfCNCPoint1[14435] = {X 463.5178, Y 44.1738, Z -1.3333, A 0.000, B 0.000, C 0.000 }
gfCNCPoint1[14436] = {X 463.5179, Y 45.0000, Z -1.3333, A 0.000, B 0.000, C 0.000 }
gfCNCPoint1[14437] = {X 463.4156, Y 45.9079, Z -1.3333, A 0.000, B 0.000, C 0.000 }
gfCNCPoint1[14438] = {X 463.1139, Y 46.7702, Z -1.3333, A 0.000, B 0.000, C 0.000 }
gfCNCPoint1[14439] = {X 462.6278, Y 47.5438, Z -1.3333, A 0.000, B 0.000, C 0.000 }
gfCNCPoint1[14440] = {X 461.9818, Y 48.1899, Z -1.3333, A 0.000, B 0.000, C 0.000 }
gfCNCPoint1[14441] = {X 461.2082, Y 48.6760, Z -1.3333, A 0.000, B 0.000, C 0.000 }
gfCNCPoint1[14442] = {X 460.3458, Y 48.9777, Z -1.3333, A 0.000, B 0.000, C 0.000 }
gfCNCPoint1[14443] = {X 459.4379, Y 49.0800, Z -1.3333, A 0.000, B 0.000, C 0.000 }
gfCNCPoint1[14444] = {X 452.9945, Y 49.0800, Z -1.3333, A 0.000, B 0.000, C 0.000 }
gfCNCPoint1[14445] = {X 452.0912, Y 48.9788, Z -1.3333, A 0.000, B 0.000, C 0.000 }
gfCNCPoint1[14446] = {X 451.2327, Y 48.6800, Z -1.3333, A 0.000, B 0.000, C 0.000 }
gfCNCPoint1[14447] = {X 450.4617, Y 48.1987, Z -1.3333, A 0.000, B 0.000, C 0.000 }
gfCNCPoint1[14448] = {X 449.8164, Y 47.5585, Z -1.3333, A 0.000, B 0.000, C 0.000 }
gfCNCPoint1[14449] = {X 449.3288, Y 46.7914, Z -1.3333, A 0.000, B 0.000, C 0.000 }
gfCNCPoint1[14450] = {X 449.0232, Y 45.9354, Z -1.3333, A 0.000, B 0.000, C 0.000 }
gfCNCPoint1[14451] = {X 448.9146, Y 45.0330, Z -1.3333, A 0.000, B 0.000, C 0.000 }
gfCNCPoint1[14452] = {X 448.9149, Y 44.1527, Z -1.3333, A 0.000, B 0.000, C 0.000 }
gfCNCPoint1[14453] = {X 449.0254, Y 43.2637, Z -1.3333, A 0.000, B 0.000, C 0.000 }
gfCNCPoint1[14454] = {X 449.3274, Y 42.4203, Z -1.3333, A 0.000, B 0.000, C 0.000 }
gfCNCPoint1[14455] = {X 449.8061, Y 41.6631, Z -1.3333, A 0.000, B 0.000, C 0.000 }
